C03646=1209.159,-22.656,-41.537,-179.909,5.502,148.937
C03647=1209.154,-22.387,-41.552,-179.907,5.502,148.936
C03648=1209.149,-22.137,-41.565,-179.904,5.503,148.936
C03649=1209.144,-21.888,-41.578,-179.901,5.503,148.935
C03650=1209.139,-21.638,-41.590,-179.899,5.503,148.934
C03651=1209.134,-21.388,-41.605,-179.897,5.503,148.934
C03652=1209.128,-21.139,-41.617,-179.894,5.504,148.933
C03653=1209.123,-20.889,-41.631,-179.891,5.504,148.932
C03654=1209.118,-20.640,-41.644,-179.889,5.504,148.932
C03655=1209.113,-20.390,-41.658,-179.887,5.505,148.931
C03656=1209.108,-20.140,-41.670,-179.884,5.505,148.930
C03657=1209.103,-19.890,-41.684,-179.882,5.506,148.930
C03658=1209.098,-19.641,-41.697,-179.880,5.505,148.929
C03659=1209.092,-19.392,-41.710,-179.877,5.506,148.928
C03660=1209.088,-19.142,-41.723,-179.874,5.506,148.928
C03661=1209.082,-18.893,-41.737,-179.872,5.507,148.927
C03662=1209.077,-18.643,-41.750,-179.870,5.507,148.926
C03663=1209.072,-18.393,-41.764,-179.867,5.507,148.926
C03664=1209.067,-18.144,-41.777,-179.864,5.508,148.925
C03665=1209.062,-17.894,-41.790,-179.862,5.508,148.924
C03666=1209.057,-17.644,-41.803,-179.860,5.508,148.924
C03667=1209.051,-17.395,-41.817,-179.857,5.509,148.923
C03668=1209.047,-17.145,-41.830,-179.855,5.509,148.922
C03669=1209.041,-16.896,-41.844,-179.852,5.510,148.922
C03670=1209.037,-16.646,-41.857,-179.850,5.509,148.921
C03671=1209.031,-16.396,-41.870,-179.847,5.510,148.920
C03672=1209.027,-16.147,-41.884,-179.845,5.510,148.920
C03673=1209.021,-15.897,-41.897,-179.842,5.511,148.919
C03674=1209.017,-15.648,-41.911,-179.840,5.510,148.918
C03675=1209.011,-15.398,-41.924,-179.838,5.511,148.918
C03676=1209.006,-15.149,-41.938,-179.835,5.512,148.917
C03677=1209.001,-14.899,-41.951,-179.832,5.512,148.916
C03678=1208.996,-14.650,-41.965,-179.830,5.512,148.916
C03679=1208.991,-14.400,-41.978,-179.828,5.512,148.915
C03680=1208.985,-14.150,-41.991,-179.825,5.513,148.914
C03681=1208.980,-13.900,-42.006,-179.822,5.513,148.914
C03682=1208.975,-13.651,-42.018,-179.820,5.514,148.913
C03683=1208.970,-13.401,-42.033,-179.818,5.514,148.912
C03684=1208.966,-13.153,-42.046,-179.815,5.514,148.911
C03685=1208.960,-12.902,-42.059,-179.813,5.515,148.911
C03686=1208.955,-12.653,-42.073,-179.810,5.515,148.910
C03687=1208.950,-12.403,-42.086,-179.808,5.515,148.910
C03688=1208.945,-12.153,-42.101,-179.805,5.516,148.909
C03689=1208.939,-11.904,-42.114,-179.803,5.516,148.908
C03690=1208.935,-11.654,-42.127,-179.800,5.517,148.908
C03691=1208.929,-11.405,-42.141,-179.798,5.517,148.907
C03692=1208.924,-11.155,-42.155,-179.795,5.517,148.906
C03693=1208.920,-10.906,-42.169,-179.793,5.517,148.905
C03694=1208.914,-10.656,-42.182,-179.791,5.518,148.905
C03695=1208.909,-10.406,-42.196,-179.788,5.519,148.904
C03696=1208.904,-10.157,-42.209,-179.785,5.519,148.904
C03697=1208.899,-9.907,-42.223,-179.783,5.519,148.903
C03698=1208.894,-9.658,-42.237,-179.781,5.519,148.902
C03699=1208.889,-9.408,-42.250,-179.778,5.520,148.902
C03700=1208.884,-9.159,-42.264,-179.775,5.520,148.901
C03701=1208.878,-8.909,-42.277,-179.773,5.520,148.900
C03702=1208.874,-8.660,-42.291,-179.771,5.520,148.899
C03703=1208.869,-8.410,-42.305,-179.768,5.521,148.899
C03704=1208.863,-8.160,-42.318,-179.766,5.522,148.898
C03705=1208.858,-7.911,-42.333,-179.763,5.522,148.898
C03706=1208.854,-7.661,-42.346,-179.761,5.522,148.897
C03707=1208.849,-7.412,-42.360,-179.758,5.522,148.896
C03708=1208.843,-7.162,-42.374,-179.756,5.523,148.896
C03709=1208.839,-6.912,-42.388,-179.753,5.523,148.895
C03710=1208.834,-6.663,-42.401,-179.750,5.524,148.894
C03711=1208.828,-6.413,-42.415,-179.748,5.524,148.893
C03712=1208.823,-6.163,-42.429,-179.746,5.524,148.893
C03713=1208.818,-5.914,-42.443,-179.743,5.525,148.892
C03714=1208.814,-5.665,-42.457,-179.741,5.525,148.892
C03715=1208.808,-5.415,-42.470,-179.738,5.526,148.891
C03716=1208.803,-5.166,-42.484,-179.736,5.526,148.890
C03717=1208.798,-4.916,-42.499,-179.733,5.526,148.890
C03718=1208.793,-4.666,-42.513,-179.731,5.527,148.889
C03719=1208.788,-4.417,-42.526,-179.728,5.527,148.888
C03720=1208.783,-4.167,-42.540,-179.725,5.528,148.887
C03721=1208.778,-3.917,-42.554,-179.723,5.529,148.887
C03722=1208.772,-3.668,-42.568,-179.721,5.528,148.886
C03723=1208.767,-3.419,-42.582,-179.719,5.529,148.886
C03724=1208.763,-3.169,-42.596,-179.716,5.529,148.885
C03725=1208.757,-2.920,-42.609,-179.713,5.530,148.884
C03726=1208.752,-2.670,-42.623,-179.711,5.530,148.884
C03727=1208.747,-2.420,-42.638,-179.709,5.530,148.883
C03728=1208.742,-2.171,-42.652,-179.706,5.530,148.882
C03729=1208.737,-1.922,-42.666,-179.703,5.531,148.882
C03730=1208.732,-1.672,-42.680,-179.701,5.532,148.881
C03731=1208.728,-1.422,-42.694,-179.698,5.532,148.880
C03732=1208.723,-1.173,-42.708,-179.696,5.533,148.880
C03733=1208.717,-0.923,-42.721,-179.694,5.532,148.879
C03734=1208.712,-0.673,-42.736,-179.691,5.533,148.878
C03735=1208.707,-0.424,-42.750,-179.688,5.533,148.878
C03736=1208.701,-0.175,-42.764,-179.686,5.534,148.877
C03737=1208.696,0.075,-42.778,-179.683,5.534,148.876
C03738=1208.691,0.325,-42.792,-179.681,5.535,148.876
C03739=1208.687,0.574,-42.807,-179.679,5.535,148.875
C03740=1208.682,0.824,-42.821,-179.676,5.536,148.874
C03741=1208.676,1.073,-42.835,-179.674,5.536,148.874
C03742=1208.672,1.323,-42.849,-179.671,5.537,148.873
C03743=1208.667,1.572,-42.863,-179.668,5.537,148.872
C03744=1208.662,1.822,-42.877,-179.666,5.538,148.872
C03745=1208.656,2.071,-42.891,-179.663,5.537,148.871
C03746=1208.651,2.321,-42.905,-179.661,5.538,148.870
C03747=1208.646,2.570,-42.920,-179.659,5.539,148.870
C03748=1208.641,2.840,-42.935,-179.656,5.539,148.869
C03749=1208.636,3.109,-42.950,-179.653,5.539,148.868
C03750=1208.629,3.378,-42.965,-179.650,5.540,148.868
C03751=1208.624,3.646,-42.981,-179.648,5.540,148.867
C03752=1208.619,3.896,-42.995,-179.645,5.541,148.866
C03753=1208.614,4.146,-43.010,-179.642,5.541,148.865
C03754=1208.609,4.396,-43.024,-179.640,5.542,148.865
C03755=1208.604,4.645,-43.038,-179.638,5.542,148.864
C03756=1208.599,4.894,-43.052,-179.635,5.542,148.864
C03757=1208.594,5.144,-43.066,-179.633,5.543,148.863
C03758=1208.589,5.394,-43.081,-179.630,5.543,148.862
C03759=1208.584,5.643,-43.095,-179.627,5.544,148.862
C03760=1208.579,5.893,-43.109,-179.625,5.544,148.861
C03761=1208.574,6.142,-43.124,-179.623,5.544,148.860
C03762=1208.569,6.391,-43.138,-179.621,5.545,148.860
C03763=1208.564,6.641,-43.152,-179.618,5.545,148.859
C03764=1208.559,6.891,-43.167,-179.615,5.546,148.858
C03765=1208.554,7.140,-43.181,-179.613,5.546,148.858
C03766=1208.549,7.390,-43.195,-179.610,5.547,148.857
C03767=1208.544,7.639,-43.210,-179.607,5.547,148.856
C03768=1208.539,7.889,-43.225,-179.605,5.548,148.856
C03769=1208.534,8.139,-43.239,-179.603,5.548,148.855
C03770=1208.529,8.388,-43.253,-179.600,5.549,148.854
C03771=1208.523,8.638,-43.268,-179.598,5.549,148.854
C03772=1208.518,8.887,-43.283,-179.595,5.550,148.853
C03773=1208.513,9.136,-43.297,-179.592,5.550,148.852
C03774=1208.508,9.386,-43.311,-179.590,5.551,148.852
C03775=1208.503,9.636,-43.325,-179.587,5.551,148.851
C03776=1208.498,9.886,-43.340,-179.585,5.551,148.850
C03777=1208.494,10.135,-43.355,-179.583,5.552,148.850
C03778=1208.489,10.384,-43.369,-179.580,5.552,148.849
C03779=1208.483,10.634,-43.384,-179.578,5.553,148.849
C03780=1208.478,10.883,-43.399,-179.575,5.553,148.848
C03781=1208.473,11.132,-43.413,-179.572,5.554,148.847
C03782=1208.468,11.382,-43.427,-179.570,5.554,148.846
C03783=1208.463,11.632,-43.441,-179.567,5.555,148.846
C03784=1208.458,11.881,-43.456,-179.565,5.555,148.845
C03785=1208.453,12.131,-43.471,-179.563,5.555,148.845
C03786=1208.448,12.381,-43.485,-179.560,5.556,148.844
C03787=1208.443,12.630,-43.500,-179.557,5.556,148.843
C03788=1208.438,12.880,-43.515,-179.555,5.557,148.843
C03789=1208.433,13.129,-43.529,-179.552,5.557,148.842
C03790=1208.428,13.379,-43.545,-179.550,5.558,148.841
C03791=1208.423,13.628,-43.559,-179.547,5.558,148.841
C03792=1208.418,13.878,-43.573,-179.545,5.559,148.840
C03793=1208.413,14.127,-43.588,-179.543,5.559,148.839
C03794=1208.408,14.377,-43.603,-179.540,5.560,148.839
C03795=1208.402,14.626,-43.618,-179.537,5.560,148.838
C03796=1208.397,14.875,-43.632,-179.535,5.561,148.837
C03797=1208.392,15.125,-43.646,-179.532,5.561,148.837
C03798=1208.387,15.374,-43.662,-179.529,5.562,148.836
C03799=1208.382,15.624,-43.676,-179.527,5.562,148.836
C03800=1208.377,15.873,-43.691,-179.525,5.563,148.835
C03801=1208.372,16.123,-43.705,-179.522,5.563,148.834
C03802=1208.367,16.372,-43.721,-179.519,5.564,148.833
C03803=1208.362,16.622,-43.735,-179.517,5.564,148.833
C03804=1208.357,16.871,-43.750,-179.515,5.564,148.832
C03805=1208.353,17.121,-43.764,-179.512,5.565,148.832
C03806=1208.347,17.370,-43.780,-179.510,5.566,148.831
C03807=1208.342,17.620,-43.794,-179.507,5.566,148.830
C03808=1208.338,17.869,-43.809,-179.504,5.567,148.830
C03809=1208.332,18.119,-43.824,-179.502,5.567,148.829
C03810=1208.327,18.368,-43.839,-179.499,5.568,148.828
C03811=1208.323,18.619,-43.854,-179.497,5.568,148.828
C03812=1208.317,18.868,-43.869,-179.494,5.569,148.827
C03813=1208.312,19.118,-43.884,-179.492,5.570,148.826
C03814=1208.308,19.367,-43.899,-179.490,5.569,148.826
C03815=1208.302,19.617,-43.914,-179.487,5.570,148.825
C03816=1208.297,19.866,-43.929,-179.484,5.570,148.824
C03817=1208.292,20.116,-43.943,-179.482,5.571,148.824
C03818=1208.287,20.365,-43.958,-179.480,5.572,148.823
C03819=1208.282,20.614,-43.973,-179.477,5.572,148.823
C03820=1208.277,20.864,-43.988,-179.474,5.573,148.822
C03821=1208.272,21.113,-44.003,-179.472,5.573,148.821
C03822=1208.267,21.363,-44.018,-179.469,5.574,148.821
C03823=1208.262,21.612,-44.033,-179.466,5.574,148.820
C03824=1208.257,21.861,-44.048,-179.464,5.575,148.819
C03825=1208.251,22.111,-44.063,-179.462,5.576,148.819
C03826=1208.247,22.361,-44.078,-179.459,5.576,148.818
C03827=1208.243,22.610,-44.093,-179.457,5.576,148.817
C03828=1208.237,22.860,-44.108,-179.454,5.577,148.817
C03829=1208.232,23.109,-44.123,-179.452,5.577,148.816
C03830=1208.227,23.359,-44.139,-179.449,5.578,148.815
C03831=1208.222,23.609,-44.153,-179.447,5.578,148.815
C03832=1208.217,23.858,-44.169,-179.444,5.579,148.814
C03833=1208.212,24.107,-44.184,-179.441,5.579,148.814
C03834=1208.207,24.356,-44.199,-179.439,5.580,148.813
C03835=1208.202,24.606,-44.214,-179.436,5.581,148.812
C03836=1208.197,24.856,-44.230,-179.433,5.581,148.811
C03837=1208.192,25.105,-44.245,-179.431,5.582,148.811
C03838=1208.187,25.355,-44.260,-179.429,5.582,148.810
C03839=1208.182,25.604,-44.274,-179.426,5.583,148.810
C03840=1208.177,25.854,-44.290,-179.423,5.584,148.809
C03841=1208.172,26.103,-44.305,-179.421,5.584,148.808
C03842=1208.167,26.352,-44.321,-179.418,5.585,148.808
C03843=1208.162,26.603,-44.335,-179.417,5.585,148.807
C03844=1208.157,26.852,-44.351,-179.414,5.585,148.806
C03845=1208.152,27.101,-44.366,-179.411,5.586,148.806
C03846=1208.147,27.351,-44.381,-179.409,5.586,148.805
C03847=1208.142,27.600,-44.396,-179.406,5.587,148.804
C03848=1208.136,27.850,-44.411,-179.403,5.587,148.804
C03849=1208.132,28.099,-44.426,-179.401,5.588,148.803
C03850=1208.127,28.349,-44.442,-179.398,5.589,148.803
C03851=1208.122,28.598,-44.457,-179.396,5.589,148.802
C03852=1208.117,28.867,-44.474,-179.393,5.590,148.801
C03853=1208.111,29.136,-44.490,-179.391,5.590,148.801
C03854=1208.106,29.404,-44.507,-179.388,5.591,148.800
C03855=1208.100,29.673,-44.523,-179.385,5.592,148.799
C03856=1208.095,29.922,-44.539,-179.382,5.593,148.799
C03857=1208.091,30.172,-44.554,-179.379,5.593,148.798
C03858=1208.085,30.421,-44.570,-179.377,5.593,148.797
C03859=1208.081,30.671,-44.585,-179.375,5.594,148.797
C03860=1208.075,30.920,-44.600,-179.373,5.594,148.796
C03861=1208.070,31.169,-44.616,-179.370,5.595,148.795
C03862=1208.066,31.419,-44.631,-179.367,5.595,148.795
C03863=1208.061,31.669,-44.647,-179.365,5.596,148.794
C03864=1208.055,31.918,-44.662,-179.362,5.596,148.793
C03865=1208.050,32.167,-44.677,-179.360,5.597,148.793
C03866=1208.046,32.417,-44.693,-179.357,5.598,148.792
C03867=1208.041,32.666,-44.708,-179.355,5.598,148.792
C03868=1208.036,32.916,-44.724,-179.352,5.599,148.791
C03869=1208.030,33.165,-44.740,-179.349,5.599,148.790
C03870=1208.026,33.415,-44.755,-179.347,5.600,148.790
C03871=1208.021,33.664,-44.770,-179.344,5.601,148.789
C03872=1208.015,33.914,-44.786,-179.342,5.601,148.788
C03873=1208.010,34.163,-44.802,-179.339,5.602,148.788
C03874=1208.006,34.413,-44.817,-179.337,5.602,148.787
C03875=1208.001,34.662,-44.833,-179.334,5.603,148.786
C03876=1207.995,34.912,-44.848,-179.332,5.604,148.786
C03877=1207.991,35.161,-44.863,-179.329,5.604,148.785
C03878=1207.986,35.411,-44.879,-179.326,5.605,148.785
C03879=1207.980,35.660,-44.895,-179.324,5.605,148.784
C03880=1207.975,35.910,-44.910,-179.321,5.606,148.783
C03881=1207.971,36.159,-44.926,-179.319,5.607,148.783
C03882=1207.966,36.408,-44.942,-179.316,5.607,148.782
C03883=1207.961,36.658,-44.958,-179.314,5.608,148.781
C03884=1207.956,36.908,-44.974,-179.311,5.608,148.781
C03885=1207.951,37.157,-44.989,-179.308,5.609,148.780
C03886=1207.946,37.406,-45.004,-179.306,5.610,148.780
C03887=1207.941,37.656,-45.020,-179.304,5.610,148.779
C03888=1207.936,37.906,-45.036,-179.301,5.611,148.778
C03889=1207.931,38.154,-45.051,-179.298,5.612,148.778
C03890=1207.926,38.404,-45.067,-179.296,5.612,148.777
C03891=1207.921,38.654,-45.083,-179.294,5.613,148.777
C03892=1207.916,38.903,-45.098,-179.291,5.613,148.776
C03893=1207.910,39.153,-45.114,-179.288,5.614,148.775
C03894=1207.906,39.402,-45.131,-179.286,5.615,148.775
C03895=1207.901,39.651,-45.146,-179.283,5.615,148.774
C03896=1207.896,39.901,-45.162,-179.281,5.616,148.773
C03897=1207.891,40.151,-45.177,-179.278,5.617,148.773
C03898=1207.886,40.399,-45.194,-179.276,5.617,148.772
C03899=1207.881,40.650,-45.210,-179.273,5.618,148.771
C03900=1207.876,40.899,-45.225,-179.270,5.618,148.771
C03901=1207.871,41.148,-45.240,-179.268,5.619,148.770
C03902=1207.867,41.397,-45.257,-179.265,5.620,148.770
C03903=1207.861,41.647,-45.272,-179.263,5.620,148.769
C03904=1207.856,41.897,-45.288,-179.260,5.621,148.768
C03905=1207.851,42.146,-45.305,-179.258,5.622,148.768
C03906=1207.846,42.395,-45.320,-179.255,5.622,148.767
C03907=1207.841,42.645,-45.336,-179.253,5.623,148.766
C03908=1207.836,42.894,-45.352,-179.250,5.623,148.766
C03909=1207.831,43.144,-45.368,-179.248,5.624,148.765
C03910=1207.827,43.393,-45.383,-179.245,5.625,148.765
C03911=1207.822,43.642,-45.400,-179.243,5.625,148.764
C03912=1207.817,43.892,-45.416,-179.240,5.626,148.763
C03913=1207.811,44.142,-45.431,-179.237,5.627,148.763
C03914=1207.807,44.391,-45.448,-179.234,5.628,148.762
C03915=1207.801,44.640,-45.464,-179.232,5.628,148.762
C03916=1207.796,44.889,-45.480,-179.229,5.629,148.761
C03917=1207.792,45.139,-45.496,-179.227,5.630,148.760
C03918=1207.786,45.389,-45.511,-179.224,5.630,148.760
C03919=1207.782,45.638,-45.528,-179.222,5.631,148.759
C03920=1207.776,45.888,-45.544,-179.219,5.632,148.758
C03921=1207.772,46.137,-45.560,-179.217,5.632,148.758
C03922=1207.767,46.386,-45.576,-179.214,5.633,148.757
C03923=1207.762,46.636,-45.593,-179.211,5.633,148.756
C03924=1207.757,46.885,-45.608,-179.209,5.634,148.756
C03925=1207.752,47.135,-45.625,-179.207,5.635,148.755
C03926=1207.747,47.384,-45.640,-179.204,5.635,148.755
C03927=1207.742,47.633,-45.657,-179.201,5.636,148.754
C03928=1207.737,47.883,-45.673,-179.199,5.637,148.753
C03929=1207.732,48.132,-45.689,-179.197,5.637,148.753
C03930=1207.727,48.382,-45.705,-179.194,5.638,148.752
C03931=1207.722,48.631,-45.721,-179.191,5.638,148.751
C03932=1207.717,48.881,-45.737,-179.189,5.639,148.751
C03933=1207.712,49.130,-45.753,-179.187,5.640,148.750
C03934=1207.707,49.380,-45.769,-179.183,5.641,148.750
C03935=1207.702,49.629,-45.786,-179.181,5.642,148.749
C03936=1207.698,49.878,-45.802,-179.179,5.642,148.749
C03937=1207.693,50.128,-45.818,-179.176,5.643,148.748
C03938=1207.688,50.377,-45.835,-179.173,5.644,148.747
C03939=1207.682,50.627,-45.851,-179.171,5.644,148.747
C03940=1207.677,50.876,-45.868,-179.168,5.645,148.746
C03941=1207.673,51.126,-45.884,-179.166,5.646,148.745
C03942=1207.667,51.375,-45.900,-179.163,5.646,148.745
C03943=1207.663,51.625,-45.916,-179.161,5.647,148.744
C03944=1207.658,51.873,-45.933,-179.158,5.647,148.743
C03945=1207.653,52.123,-45.949,-179.156,5.648,148.743
C03946=1207.648,52.372,-45.965,-179.153,5.649,148.742
C03947=1207.644,52.622,-45.982,-179.151,5.649,148.742
C03948=1207.637,52.871,-45.998,-179.147,5.651,148.741
C03949=1207.633,53.121,-46.015,-179.145,5.651,148.741
C03950=1207.628,53.370,-46.031,-179.143,5.652,148.740
C03951=1207.623,53.620,-46.047,-179.140,5.653,148.739
C03952=1207.619,53.869,-46.063,-179.137,5.653,148.739
C03953=1207.613,54.118,-46.080,-179.135,5.654,148.738
C03954=1207.608,54.368,-46.097,-179.132,5.655,148.737
C03955=1207.603,54.617,-46.113,-179.130,5.655,148.737
C03956=1207.598,54.886,-46.131,-179.127,5.656,148.736
C03957=1207.593,55.154,-46.148,-179.124,5.657,148.735
C03958=1207.588,55.423,-46.166,-179.121,5.658,148.735
C03959=1207.582,55.691,-46.184,-179.119,5.658,148.734
C03960=1207.577,55.941,-46.200,-179.117,5.659,148.734
C03961=1207.572,56.190,-46.216,-179.114,5.660,148.733
C03962=1207.568,56.439,-46.233,-179.111,5.660,148.732
C03963=1207.562,56.689,-46.250,-179.109,5.661,148.732
C03964=1207.557,56.938,-46.267,-179.106,5.662,148.731
C03965=1207.553,57.187,-46.283,-179.103,5.663,148.731
C03966=1207.548,57.437,-46.299,-179.101,5.663,148.730
C03967=1207.542,57.687,-46.316,-179.098,5.664,148.729
C03968=1207.538,57.936,-46.333,-179.096,5.665,148.729
C03969=1207.533,58.185,-46.349,-179.093,5.665,148.728
C03970=1207.528,58.434,-46.366,-179.091,5.666,148.728
C03971=1207.523,58.684,-46.383,-179.088,5.667,148.727
C03972=1207.518,58.933,-46.399,-179.086,5.667,148.726
C03973=1207.513,59.182,-46.416,-179.083,5.669,148.726
C03974=1207.508,59.433,-46.433,-179.080,5.669,148.725
C03975=1207.503,59.682,-46.449,-179.078,5.670,148.725
C03976=1207.498,59.931,-46.466,-179.075,5.671,148.724
C03977=1207.493,60.181,-46.483,-179.073,5.671,148.723
C03978=1207.488,60.430,-46.499,-179.070,5.672,148.723
C03979=1207.484,60.679,-46.516,-179.068,5.673,148.722
C03980=1207.478,60.929,-46.533,-179.065,5.673,148.722
C03981=1207.473,61.178,-46.549,-179.063,5.674,148.721
C03982=1207.469,61.427,-46.566,-179.060,5.676,148.720
C03983=1207.464,61.677,-46.583,-179.057,5.676,148.720
C03984=1207.459,61.926,-46.600,-179.055,5.677,148.719
C03985=1207.454,62.175,-46.616,-179.052,5.677,148.718
C03986=1207.449,62.425,-46.634,-179.050,5.678,148.718
C03987=1207.444,62.675,-46.650,-179.047,5.679,148.717
C03988=1207.439,62.924,-46.667,-179.045,5.679,148.717
C03989=1207.434,63.173,-46.684,-179.042,5.681,148.716
C03990=1207.430,63.423,-46.700,-179.039,5.682,148.716
C03991=1207.424,63.672,-46.717,-179.037,5.682,148.715
C03992=1207.419,63.921,-46.734,-179.034,5.683,148.714
C03993=1207.414,64.171,-46.751,-179.032,5.684,148.714
C03994=1207.410,64.420,-46.769,-179.029,5.684,148.713
C03995=1207.405,64.669,-46.785,-179.027,5.685,148.713
C03996=1207.400,64.918,-46.802,-179.024,5.686,148.712
C03997=1207.395,65.168,-46.819,-179.021,5.687,148.711
C03998=1207.390,65.418,-46.836,-179.019,5.688,148.711
C03999=1207.385,65.667,-46.852,-179.016,5.688,148.710
C04000=1207.380,65.916,-46.870,-179.014,5.689,148.710
C04001=1207.375,66.166,-46.886,-179.011,5.690,148.709
C04002=1207.370,66.415,-46.904,-179.008,5.690,148.708
C04003=1207.366,66.664,-46.921,-179.006,5.692,148.708
C04004=1207.361,66.913,-46.937,-179.003,5.693,148.707
C04005=1207.355,67.163,-46.955,-179.001,5.693,148.707
C04006=1207.351,67.413,-46.971,-178.998,5.694,148.706
C04007=1207.346,67.662,-46.989,-178.996,5.695,148.706
C04008=1207.342,67.911,-47.006,-178.993,5.695,148.705
C04009=1207.336,68.160,-47.023,-178.990,5.696,148.704
C04010=1207.331,68.410,-47.039,-178.988,5.697,148.704
C04011=1207.326,68.660,-47.057,-178.985,5.698,148.703
C04012=1207.321,68.909,-47.075,-178.982,5.699,148.702
C04013=1207.317,69.158,-47.091,-178.980,5.699,148.702
C04014=1207.311,69.407,-47.108,-178.978,5.700,148.701
C04015=1207.306,69.657,-47.125,-178.975,5.701,148.701
C04016=1207.301,69.906,-47.143,-178.972,5.702,148.700
C04017=1207.297,70.155,-47.160,-178.970,5.703,148.700
C04018=1207.292,70.405,-47.177,-178.967,5.703,148.699
C04019=1207.288,70.654,-47.194,-178.965,5.704,148.698
C04020=1207.282,70.903,-47.211,-178.962,5.705,148.698
C04021=1207.277,71.153,-47.228,-178.960,5.705,148.697
C04022=1207.272,71.402,-47.246,-178.957,5.707,148.697
C04023=1207.267,71.652,-47.263,-178.954,5.708,148.696
C04024=1207.263,71.901,-47.280,-178.952,5.708,148.695
C04025=1207.258,72.150,-47.298,-178.949,5.709,148.695
C04026=1207.253,72.400,-47.315,-178.947,5.710,148.694
C04027=1207.248,72.650,-47.332,-178.944,5.711,148.694
C04028=1207.243,72.898,-47.349,-178.941,5.712,148.693
C04029=1207.237,73.148,-47.367,-178.939,5.713,148.693
C04030=1207.233,73.397,-47.384,-178.936,5.713,148.692
C04031=1207.228,73.647,-47.401,-178.934,5.714,148.691
C04032=1207.223,73.896,-47.418,-178.931,5.716,148.691
C04033=1207.219,74.145,-47.436,-178.928,5.716,148.690
C04034=1207.213,74.395,-47.453,-178.926,5.717,148.690
C04035=1207.208,74.644,-47.471,-178.924,5.718,148.689
C04036=1207.204,74.894,-47.488,-178.921,5.718,148.688
C04037=1207.198,75.142,-47.505,-178.918,5.719,148.688
C04038=1207.193,75.392,-47.523,-178.916,5.720,148.687
C04039=1207.189,75.641,-47.540,-178.913,5.721,148.687
C04040=1207.184,75.891,-47.557,-178.910,5.722,148.686
C04041=1207.179,76.140,-47.575,-178.908,5.723,148.686
C04042=1207.174,76.389,-47.592,-178.906,5.723,148.685
C04043=1207.169,76.638,-47.610,-178.902,5.724,148.684
C04044=1207.164,76.888,-47.627,-178.900,5.725,148.684
C04045=1207.159,77.137,-47.645,-178.898,5.726,148.683
C04046=1207.155,77.387,-47.662,-178.895,5.727,148.683
C04047=1207.150,77.636,-47.680,-178.892,5.728,148.682
C04048=1207.145,77.885,-47.698,-178.890,5.729,148.681
C04049=1207.140,78.135,-47.715,-178.887,5.729,148.681
C04050=1207.136,78.384,-47.732,-178.885,5.730,148.680
C04051=1207.130,78.634,-47.750,-178.882,5.731,148.680
C04052=1207.126,78.883,-47.768,-178.879,5.732,148.679
C04053=1207.121,79.132,-47.786,-178.877,5.733,148.679
C04054=1207.115,79.382,-47.803,-178.874,5.734,148.678
C04055=1207.111,79.631,-47.820,-178.872,5.735,148.678
C04056=1207.106,79.881,-47.838,-178.869,5.736,148.677
C04057=1207.101,80.130,-47.856,-178.866,5.737,148.676
C04058=1207.096,80.379,-47.874,-178.864,5.738,148.676
C04059=1207.091,80.629,-47.891,-178.862,5.738,148.675
C04060=1207.085,80.896,-47.910,-178.858,5.740,148.675
C04061=1207.080,81.164,-47.929,-178.856,5.740,148.674
C04062=1207.076,81.433,-47.947,-178.853,5.741,148.673
C04063=1207.070,81.701,-47.967,-178.850,5.742,148.673
C04064=1207.065,81.951,-47.984,-178.848,5.743,148.672
C04065=1207.060,82.200,-48.002,-178.845,5.744,148.672
C04066=1207.055,82.449,-48.020,-178.843,5.745,148.671
C04067=1207.051,82.699,-48.038,-178.840,5.746,148.670
C04068=1207.045,82.948,-48.055,-178.837,5.746,148.670
C04069=1207.040,83.198,-48.073,-178.835,5.747,148.669
C04070=1207.035,83.447,-48.091,-178.833,5.748,148.669
C04071=1207.031,83.696,-48.109,-178.829,5.749,148.668
C04072=1207.026,83.945,-48.127,-178.827,5.750,148.668
C04073=1207.021,84.195,-48.144,-178.825,5.751,148.667
C04074=1207.017,84.444,-48.162,-178.822,5.752,148.667
C04075=1207.012,84.694,-48.180,-178.819,5.753,148.666
C04076=1207.007,84.943,-48.198,-178.817,5.754,148.665
C04077=1207.002,85.192,-48.216,-178.814,5.755,148.665
C04078=1206.997,85.442,-48.233,-178.812,5.755,148.664
C04079=1206.992,85.691,-48.251,-178.809,5.757,148.664
C04080=1206.987,85.940,-48.269,-178.807,5.758,148.663
C04081=1206.982,86.189,-48.287,-178.804,5.758,148.662
C04082=1206.977,86.438,-48.305,-178.801,5.760,148.662
C04083=1206.972,86.688,-48.323,-178.799,5.760,148.661
C04084=1206.967,86.937,-48.341,-178.796,5.761,148.661
C04085=1206.963,87.187,-48.360,-178.794,5.762,148.660
C04086=1206.958,87.436,-48.378,-178.791,5.763,148.660
C04087=1206.953,87.685,-48.396,-178.788,5.764,148.659
C04088=1206.948,87.935,-48.413,-178.786,5.765,148.659
C04089=1206.943,88.184,-48.431,-178.783,5.765,148.658
C04090=1206.938,88.433,-48.449,-178.781,5.767,148.658
C04091=1206.933,88.682,-48.467,-178.778,5.768,148.657
C04092=1206.928,88.932,-48.485,-178.776,5.769,148.656
C04093=1206.924,89.181,-48.503,-178.773,5.769,148.656
C04094=1206.919,89.431,-48.521,-178.770,5.771,148.655
C04095=1206.914,89.680,-48.539,-178.768,5.772,148.655
C04096=1206.909,89.929,-48.557,-178.765,5.772,148.654
C04097=1206.904,90.178,-48.575,-178.763,5.774,148.654
C04098=1206.900,90.427,-48.593,-178.760,5.774,148.653
C04099=1206.895,90.676,-48.611,-178.757,5.775,148.652
C04100=1206.890,90.926,-48.629,-178.755,5.776,148.652
C04101=1206.885,91.176,-48.648,-178.752,5.777,148.651
C04102=1206.880,91.424,-48.667,-178.750,5.778,148.651
C04103=1206.875,91.674,-48.685,-178.747,5.779,148.650
C04104=1206.870,91.923,-48.703,-178.744,5.780,148.650
C04105=1206.866,92.173,-48.721,-178.742,5.781,148.649
C04106=1206.861,92.422,-48.739,-178.739,5.782,148.649
C04107=1206.856,92.671,-48.757,-178.737,5.784,148.648
C04108=1206.851,92.920,-48.775,-178.734,5.784,148.647
C04109=1206.846,93.170,-48.793,-178.731,5.785,148.647
C04110=1206.841,93.420,-48.812,-178.729,5.786,148.646
C04111=1206.837,93.668,-48.830,-178.726,5.787,148.646
C04112=1206.832,93.917,-48.848,-178.724,5.788,148.645
C04113=1206.827,94.166,-48.866,-178.721,5.789,148.645
C04114=1206.822,94.416,-48.885,-178.718,5.790,148.644
C04115=1206.817,94.666,-48.903,-178.716,5.791,148.644
C04116=1206.812,94.915,-48.921,-178.713,5.791,148.643
C04117=1206.807,95.164,-48.940,-178.711,5.793,148.643
C04118=1206.802,95.413,-48.958,-178.708,5.794,148.642
C04119=1206.798,95.663,-48.976,-178.706,5.795,148.641
C04120=1206.792,95.912,-48.995,-178.703,5.796,148.641
C04121=1206.788,96.161,-49.014,-178.700,5.797,148.640
C04122=1206.783,96.410,-49.032,-178.698,5.798,148.640
C04123=1206.779,96.660,-49.050,-178.695,5.798,148.639
C04124=1206.774,96.909,-49.068,-178.693,5.800,148.639
C04125=1206.768,97.158,-49.087,-178.690,5.801,148.638
C04126=1206.764,97.408,-49.106,-178.688,5.801,148.638
C04127=1206.759,97.657,-49.124,-178.685,5.803,148.637
C04128=1206.754,97.906,-49.143,-178.682,5.804,148.637
C04129=1206.749,98.155,-49.161,-178.680,5.804,148.636
C04130=1206.745,98.405,-49.179,-178.677,5.806,148.635
C04131=1206.740,98.654,-49.197,-178.675,5.807,148.635
C04132=1206.734,98.903,-49.216,-178.672,5.807,148.634
C04133=1206.730,99.153,-49.235,-178.669,5.809,148.634
C04134=1206.725,99.401,-49.253,-178.667,5.810,148.633
C04135=1206.720,99.651,-49.272,-178.664,5.811,148.633
C04136=1206.715,99.901,-49.290,-178.661,5.812,148.632
C04137=1206.711,100.149,-49.309,-178.659,5.813,148.632
C04138=1206.705,100.399,-49.328,-178.657,5.814,148.631
C04139=1206.701,100.648,-49.347,-178.653,5.815,148.630
C04140=1206.696,100.897,-49.365,-178.651,5.816,148.630
C04141=1206.691,101.146,-49.383,-178.649,5.816,148.629
C04142=1206.687,101.396,-49.402,-178.646,5.818,148.629
C04143=1206.682,101.645,-49.420,-178.643,5.819,148.628
C04144=1206.676,101.894,-49.440,-178.641,5.821,148.628
C04145=1206.672,102.144,-49.458,-178.638,5.821,148.627
C04146=1206.667,102.392,-49.477,-178.636,5.822,148.627
C04147=1206.662,102.642,-49.495,-178.633,5.823,148.626
C04148=1206.658,102.891,-49.514,-178.631,5.824,148.626
C04149=1206.652,103.140,-49.533,-178.628,5.825,148.625
C04150=1206.648,103.390,-49.552,-178.625,5.826,148.625
C04151=1206.643,103.639,-49.570,-178.623,5.827,148.624
C04152=1206.638,103.888,-49.589,-178.620,5.828,148.623
C04153=1206.634,104.138,-49.608,-178.617,5.830,148.623
C04154=1206.628,104.386,-49.627,-178.615,5.830,148.622
C04155=1206.623,104.636,-49.645,-178.613,5.831,148.622
C04156=1206.619,104.885,-49.664,-178.609,5.833,148.621
C04157=1206.614,105.134,-49.682,-178.607,5.834,148.621
C04158=1206.609,105.384,-49.702,-178.604,5.835,148.620
C04159=1206.604,105.633,-49.721,-178.602,5.836,148.620
C04160=1206.600,105.882,-49.739,-178.599,5.837,148.619
C04161=1206.595,106.131,-49.758,-178.597,5.838,148.619
C04162=1206.590,106.380,-49.777,-178.594,5.839,148.618
C04163=1206.585,106.630,-49.796,-178.592,5.840,148.618
C04164=1206.579,106.898,-49.817,-178.589,5.841,148.617
C04165=1206.575,107.167,-49.837,-178.585,5.843,148.617
C04166=1206.569,107.435,-49.857,-178.583,5.843,148.616
C04167=1206.564,107.703,-49.877,-178.580,5.845,148.615
C04168=1206.560,107.953,-49.896,-178.578,5.846,148.615
C04169=1206.554,108.202,-49.916,-178.575,5.847,148.614
C04170=1206.550,108.451,-49.934,-178.572,5.848,148.614
C04171=1206.545,108.700,-49.953,-178.570,5.849,148.613
C04172=1206.540,108.950,-49.973,-178.567,5.850,148.613
C04173=1206.535,109.198,-49.992,-178.565,5.851,148.612
C04174=1206.530,109.449,-50.011,-178.562,5.852,148.612
C04175=1206.526,109.697,-50.029,-178.560,5.854,148.611
C04176=1206.521,109.947,-50.049,-178.557,5.854,148.611
C04177=1206.516,110.195,-50.068,-178.554,5.856,148.610
C04178=1206.511,110.445,-50.087,-178.552,5.857,148.610
C04179=1206.506,110.694,-50.106,-178.549,5.857,148.609
C04180=1206.502,110.944,-50.125,-178.546,5.859,148.609
C04181=1206.497,111.192,-50.144,-178.544,5.860,148.608
C04182=1206.493,111.442,-50.163,-178.541,5.861,148.608
C04183=1206.487,111.691,-50.182,-178.539,5.862,148.607
C04184=1206.482,111.941,-50.201,-178.536,5.864,148.606
C04185=1206.478,112.189,-50.220,-178.534,5.865,148.606
C04186=1206.473,112.439,-50.240,-178.531,5.865,148.605
C04187=1206.467,112.688,-50.259,-178.528,5.867,148.605
C04188=1206.463,112.937,-50.278,-178.526,5.868,148.604
C04189=1206.458,113.186,-50.297,-178.523,5.869,148.604
C04190=1206.453,113.435,-50.317,-178.520,5.870,148.603
C04191=1206.449,113.685,-50.335,-178.518,5.871,148.603
C04192=1206.444,113.934,-50.355,-178.515,5.872,148.602
C04193=1206.439,114.184,-50.374,-178.513,5.873,148.602
C04194=1206.434,114.432,-50.393,-178.510,5.875,148.601
C04195=1206.430,114.682,-50.413,-178.508,5.876,148.601
C04196=1206.424,114.931,-50.432,-178.504,5.877,148.600
C04197=1206.420,115.180,-50.452,-178.502,5.878,148.600
C04198=1206.416,115.430,-50.471,-178.500,5.879,148.599
C04199=1206.410,115.678,-50.490,-178.497,5.880,148.599
C04200=1206.405,115.928,-50.510,-178.495,5.881,148.598
C04201=1206.400,116.177,-50.529,-178.492,5.883,148.598
C04202=1206.396,116.426,-50.548,-178.490,5.884,148.597
C04203=1206.391,116.675,-50.567,-178.486,5.885,148.597
C04204=1206.386,116.925,-50.587,-178.484,5.886,148.596
C04205=1206.381,117.174,-50.607,-178.482,5.887,148.596
C04206=1206.377,117.423,-50.625,-178.479,5.888,148.595
C04207=1206.372,117.672,-50.645,-178.476,5.889,148.595
C04208=1206.367,117.922,-50.665,-178.474,5.891,148.594
C04209=1206.362,118.171,-50.684,-178.471,5.891,148.594
C04210=1206.357,118.420,-50.704,-178.468,5.893,148.593
C04211=1206.353,118.668,-50.723,-178.466,5.894,148.593
C04212=1206.348,118.918,-50.743,-178.463,5.895,148.592
C04213=1206.343,119.167,-50.762,-178.461,5.896,148.592
C04214=1206.338,119.416,-50.782,-178.458,5.898,148.591
C04215=1206.333,119.666,-50.801,-178.456,5.899,148.591
C04216=1206.328,119.915,-50.821,-178.453,5.899,148.590
C04217=1206.324,120.164,-50.840,-178.450,5.901,148.590
C04218=1206.319,120.413,-50.860,-178.448,5.902,148.589
C04219=1206.315,120.662,-50.880,-178.445,5.904,148.589
C04220=1206.309,120.911,-50.899,-178.442,5.904,148.588
C04221=1206.305,121.161,-50.919,-178.440,5.906,148.588
C04222=1206.300,121.410,-50.938,-178.438,5.907,148.587
C04223=1206.295,121.659,-50.958,-178.434,5.908,148.587
C04224=1206.290,121.908,-50.978,-178.432,5.909,148.586
C04225=1206.286,122.158,-50.997,-178.429,5.911,148.586
C04226=1206.281,122.406,-51.016,-178.427,5.912,148.585
C04227=1206.276,122.656,-51.036,-178.424,5.913,148.585
C04228=1206.272,122.905,-51.056,-178.422,5.914,148.584
C04229=1206.267,123.154,-51.076,-178.419,5.916,148.584
C04230=1206.261,123.403,-51.095,-178.416,5.916,148.583
C04231=1206.257,123.652,-51.116,-178.414,5.918,148.583
C04232=1206.252,123.902,-51.135,-178.411,5.919,148.582
C04233=1206.248,124.151,-51.155,-178.408,5.920,148.582
C04234=1206.242,124.400,-51.174,-178.406,5.921,148.581
C04235=1206.238,124.649,-51.195,-178.404,5.922,148.581
C04236=1206.233,124.899,-51.214,-178.401,5.924,148.580
C04237=1206.228,125.147,-51.234,-178.398,5.924,148.580
C04238=1206.223,125.397,-51.254,-178.396,5.926,148.579
C04239=1206.218,125.646,-51.274,-178.393,5.927,148.579
C04240=1206.214,125.895,-51.294,-178.390,5.929,148.578
C04241=1206.209,126.145,-51.314,-178.388,5.929,148.578
C04242=1206.204,126.394,-51.333,-178.385,5.931,148.577
C04243=1206.200,126.643,-51.353,-178.383,5.932,148.577
C04244=1206.195,126.892,-51.373,-178.380,5.933,148.576
C04245=1206.190,127.141,-51.393,-178.378,5.934,148.576
C04246=1206.185,127.390,-51.413,-178.375,5.936,148.575
C04247=1206.181,127.639,-51.433,-178.372,5.937,148.575
C04248=1206.176,127.888,-51.453,-178.370,5.938,148.574
C04249=1206.171,128.138,-51.472,-178.367,5.939,148.574
C04250=1206.167,128.387,-51.493,-178.364,5.941,148.573
C04251=1206.161,128.636,-51.512,-178.361,5.942,148.573
C04252=1206.157,128.885,-51.532,-178.359,5.943,148.572
C04253=1206.152,129.134,-51.552,-178.356,5.945,148.572
C04254=1206.148,129.383,-51.572,-178.354,5.946,148.571
C04255=1206.143,129.633,-51.593,-178.351,5.947,148.571
C04256=1206.138,129.882,-51.613,-178.349,5.948,148.570
C04257=1206.133,130.130,-51.633,-178.346,5.950,148.570
C04258=1206.128,130.380,-51.653,-178.344,5.951,148.569
C04259=1206.124,130.629,-51.673,-178.341,5.952,148.569
C04260=1206.119,130.878,-51.693,-178.338,5.953,148.568
C04261=1206.114,131.127,-51.713,-178.336,5.955,148.568
C04262=1206.109,131.377,-51.733,-178.333,5.955,148.567
C04263=1206.104,131.626,-51.753,-178.331,5.957,148.567
C04264=1206.099,131.874,-51.774,-178.328,5.958,148.566
C04265=1206.095,132.124,-51.793,-178.325,5.960,148.566
C04266=1206.090,132.373,-51.814,-178.323,5.961,148.566
C04267=1206.086,132.622,-51.834,-178.320,5.962,148.565
C04268=1206.080,132.891,-51.856,-178.317,5.964,148.565
C04269=1206.074,133.160,-51.877,-178.315,5.964,148.564
C04270=1206.070,133.428,-51.899,-178.312,5.966,148.564
C04271=1206.064,133.697,-51.921,-178.309,5.968,148.563
C04272=1206.060,133.946,-51.941,-178.307,5.969,148.563
C04273=1206.055,134.195,-51.962,-178.304,5.970,148.562
C04274=1206.051,134.444,-51.982,-178.301,5.972,148.562
C04275=1206.045,134.694,-52.002,-178.299,5.973,148.561
C04276=1206.041,134.943,-52.023,-178.296,5.974,148.561
C04277=1206.037,135.191,-52.043,-178.293,5.975,148.560
C04278=1206.032,135.441,-52.063,-178.290,5.977,148.559
C04279=1206.027,135.690,-52.084,-178.288,5.978,148.559
C04280=1206.022,135.939,-52.104,-178.285,5.979,148.559
C04281=1206.017,136.187,-52.124,-178.283,5.980,148.558
C04282=1206.012,136.437,-52.145,-178.280,5.982,148.558
C04283=1206.007,136.686,-52.165,-178.277,5.984,148.557
C04284=1206.003,136.935,-52.185,-178.275,5.984,148.557
C04285=1205.998,137.184,-52.205,-178.272,5.986,148.556
C04286=1205.993,137.433,-52.226,-178.270,5.987,148.556
C04287=1205.989,137.682,-52.247,-178.267,5.988,148.555
C04288=1205.984,137.931,-52.267,-178.265,5.989,148.555
C04289=1205.979,138.181,-52.287,-178.262,5.991,148.554
C04290=1205.974,138.430,-52.308,-178.259,5.993,148.554
C04291=1205.970,138.679,-52.328,-178.257,5.993,148.553
C04292=1205.965,138.928,-52.349,-178.254,5.995,148.553
C04293=1205.960,139.177,-52.369,-178.252,5.996,148.552
C04294=1205.955,139.427,-52.390,-178.249,5.998,148.552
C04295=1205.951,139.676,-52.411,-178.247,5.999,148.552
C04296=1205.946,139.925,-52.431,-178.244,6.000,148.551
C04297=1205.941,140.174,-52.452,-178.241,6.002,148.551
C04298=1205.937,140.423,-52.472,-178.239,6.003,148.550
C04299=1205.932,140.672,-52.493,-178.236,6.004,148.550
C04300=1205.927,140.921,-52.514,-178.234,6.005,148.549
C04301=1205.923,141.170,-52.534,-178.231,6.007,148.549
C04302=1205.917,141.419,-52.555,-178.228,6.008,148.548
C04303=1205.913,141.668,-52.576,-178.226,6.009,148.548
C04304=1205.908,141.917,-52.596,-178.223,6.011,148.548
C04305=1205.903,142.166,-52.617,-178.220,6.012,148.547
C04306=1205.898,142.416,-52.638,-178.218,6.014,148.547
C04307=1205.894,142.665,-52.658,-178.215,6.015,148.546
C04308=1205.889,142.913,-52.679,-178.212,6.016,148.545
C04309=1205.884,143.163,-52.700,-178.210,6.018,148.545
C04310=1205.880,143.412,-52.720,-178.208,6.019,148.545
C04311=1205.875,143.662,-52.741,-178.204,6.020,148.544
C04312=1205.871,143.911,-52.762,-178.202,6.022,148.544
C04313=1205.866,144.160,-52.783,-178.200,6.023,148.543
C04314=1205.861,144.409,-52.803,-178.197,6.025,148.543
C04315=1205.856,144.658,-52.824,-178.194,6.025,148.542
C04316=1205.852,144.906,-52.845,-178.192,6.027,148.542
C04317=1205.847,145.156,-52.866,-178.189,6.029,148.542
C04318=1205.842,145.405,-52.886,-178.186,6.030,148.541
C04319=1205.837,145.654,-52.907,-178.184,6.031,148.541
C04320=1205.832,145.903,-52.928,-178.181,6.033,148.540
C04321=1205.828,146.153,-52.949,-178.178,6.034,148.540
C04322=1205.823,146.401,-52.971,-178.176,6.036,148.539
C04323=1205.819,146.650,-52.991,-178.174,6.036,148.539
C04324=1205.814,146.900,-53.012,-178.171,6.038,148.538
C04325=1205.809,147.149,-53.032,-178.168,6.040,148.538
C04326=1205.804,147.397,-53.054,-178.166,6.041,148.537
C04327=1205.799,147.646,-53.075,-178.163,6.042,148.537
C04328=1205.795,147.895,-53.095,-178.160,6.044,148.536
C04329=1205.790,148.145,-53.117,-178.158,6.045,148.536
C04330=1205.786,148.394,-53.138,-178.155,6.047,148.536
C04331=1205.781,148.643,-53.159,-178.153,6.048,148.535
C04332=1205.776,148.892,-53.180,-178.150,6.049,148.535
C04333=1205.771,149.141,-53.200,-178.147,6.051,148.534
C04334=1205.766,149.390,-53.222,-178.145,6.052,148.534
C04335=1205.762,149.640,-53.243,-178.142,6.053,148.533
C04336=1205.757,149.889,-53.264,-178.139,6.055,148.533
C04337=1205.752,150.137,-53.285,-178.137,6.056,148.532
C04338=1205.747,150.387,-53.306,-178.134,6.058,148.532
C04339=1205.743,150.635,-53.327,-178.131,6.059,148.532
C04340=1205.738,150.884,-53.348,-178.129,6.060,148.531
C04341=1205.733,151.134,-53.370,-178.126,6.062,148.531
C04342=1205.729,151.382,-53.391,-178.124,6.064,148.530
C04343=1205.724,151.632,-53.412,-178.121,6.064,148.530
C04344=1205.719,151.880,-53.433,-178.118,6.066,148.529
C04345=1205.714,152.130,-53.454,-178.116,6.068,148.529
C04346=1205.710,152.379,-53.475,-178.114,6.069,148.529
C04347=1205.705,152.628,-53.497,-178.111,6.070,148.528
C04348=1205.700,152.877,-53.518,-178.108,6.072,148.528
C04349=1205.695,153.126,-53.539,-178.106,6.073,148.527
C04350=1205.691,153.375,-53.560,-178.103,6.075,148.527
C04351=1205.687,153.624,-53.582,-178.100,6.076,148.526
C04352=1205.681,153.873,-53.603,-178.098,6.077,148.526
C04353=1205.677,154.122,-53.624,-178.095,6.079,148.525
C04354=1205.673,154.372,-53.645,-178.092,6.081,148.525
C04355=1205.668,154.620,-53.667,-178.090,6.082,148.525
C04356=1205.663,154.870,-53.688,-178.087,6.083,148.524
C04357=1205.658,155.118,-53.709,-178.085,6.085,148.524
C04358=1205.653,155.368,-53.731,-178.082,6.086,148.523
C04359=1205.649,155.617,-53.752,-178.079,6.088,148.523
C04360=1205.644,155.865,-53.774,-178.077,6.089,148.522
C04361=1205.639,156.114,-53.795,-178.074,6.090,148.522
C04362=1205.635,156.364,-53.817,-178.072,6.092,148.522
C04363=1205.630,156.613,-53.838,-178.069,6.094,148.521
C04364=1205.625,156.862,-53.859,-178.067,6.095,148.521
C04365=1205.621,157.111,-53.881,-178.064,6.096,148.520
C04366=1205.616,157.360,-53.902,-178.061,6.098,148.520
C04367=1205.611,157.609,-53.923,-178.059,6.100,148.520
C04368=1205.607,157.858,-53.945,-178.056,6.101,148.519
C04369=1205.602,158.107,-53.966,-178.053,6.102,148.519
C04370=1205.597,158.356,-53.988,-178.051,6.104,148.518
C04371=1205.592,158.604,-54.010,-178.048,6.105,148.518
C04372=1205.587,158.873,-54.033,-178.045,6.107,148.517
C04373=1205.582,159.143,-54.056,-178.043,6.109,148.517
C04374=1205.577,159.411,-54.079,-178.040,6.110,148.516
C04375=1205.572,159.681,-54.103,-178.037,6.112,148.516
C04376=1205.568,159.930,-54.125,-178.034,6.114,148.515
C04377=1205.562,160.179,-54.146,-178.032,6.115,148.515
C04378=1205.557,160.428,-54.167,-178.029,6.116,148.514
C04379=1205.553,160.677,-54.189,-178.026,6.118,148.514
C04380=1205.548,160.926,-54.211,-178.024,6.120,148.514
C04381=1205.544,161.175,-54.233,-178.021,6.121,148.513
C04382=1205.539,161.424,-54.254,-178.019,6.122,148.513
C04383=1205.534,161.673,-54.276,-178.016,6.124,148.512
C04384=1205.530,161.922,-54.298,-178.013,6.126,148.512
C04385=1205.525,162.171,-54.320,-178.011,6.127,148.512
C04386=1205.521,162.420,-54.342,-178.008,6.128,148.511
C04387=1205.516,162.669,-54.363,-178.006,6.130,148.511
C04388=1205.511,162.918,-54.385,-178.003,6.131,148.510
C04389=1205.506,163.168,-54.406,-178.000,6.133,148.510
C04390=1205.501,163.416,-54.428,-177.998,6.134,148.510
C04391=1205.497,163.666,-54.450,-177.995,6.136,148.509
C04392=1205.492,163.914,-54.472,-177.993,6.137,148.509
C04393=1205.487,164.163,-54.493,-177.990,6.139,148.508
C04394=1205.483,164.412,-54.515,-177.987,6.140,148.508
C04395=1205.478,164.661,-54.537,-177.984,6.142,148.507
C04396=1205.474,164.910,-54.559,-177.982,6.143,148.507
C04397=1205.469,165.159,-54.581,-177.980,6.145,148.507
C04398=1205.465,165.408,-54.603,-177.977,6.147,148.506
C04399=1205.460,165.657,-54.625,-177.974,6.148,148.506
C04400=1205.455,165.907,-54.647,-177.972,6.149,148.505
C04401=1205.450,166.155,-54.669,-177.969,6.151,148.505
C04402=1205.446,166.405,-54.691,-177.966,6.153,148.505
C04403=1205.441,166.653,-54.713,-177.964,6.155,148.504
C04404=1205.436,166.902,-54.734,-177.962,6.156,148.504
C04405=1205.432,167.151,-54.756,-177.958,6.157,148.503
C04406=1205.427,167.400,-54.778,-177.956,6.159,148.503
C04407=1205.423,167.649,-54.800,-177.953,6.161,148.503
C04408=1205.417,167.898,-54.822,-177.951,6.162,148.502
C04409=1205.413,168.147,-54.844,-177.948,6.164,148.502
C04410=1205.408,168.396,-54.866,-177.946,6.165,148.501
C04411=1205.404,168.645,-54.889,-177.942,6.167,148.501
C04412=1205.399,168.893,-54.911,-177.940,6.169,148.500
C04413=1205.394,169.143,-54.933,-177.938,6.170,148.500
C04414=1205.389,169.392,-54.955,-177.935,6.171,148.500
C04415=1205.385,169.641,-54.977,-177.932,6.173,148.499
C04416=1205.380,169.890,-54.999,-177.930,6.175,148.499
C04417=1205.376,170.139,-55.021,-177.928,6.176,148.499
C04418=1205.371,170.388,-55.044,-177.924,6.177,148.498
C04419=1205.366,170.637,-55.066,-177.922,6.179,148.498
C04420=1205.362,170.886,-55.088,-177.919,6.181,148.497
C04421=1205.357,171.135,-55.109,-177.916,6.183,148.497
C04422=1205.352,171.384,-55.132,-177.914,6.184,148.497
C04423=1205.348,171.632,-55.154,-177.912,6.186,148.496
C04424=1205.343,171.882,-55.177,-177.909,6.187,148.496
C04425=1205.338,172.131,-55.199,-177.906,6.189,148.495
C04426=1205.334,172.379,-55.222,-177.903,6.191,148.495
C04427=1205.329,172.629,-55.244,-177.901,6.192,148.494
C04428=1205.325,172.877,-55.265,-177.898,6.193,148.494
C04429=1205.320,173.127,-55.288,-177.896,6.195,148.494
C04430=1205.315,173.375,-55.310,-177.893,6.197,148.493
C04431=1205.311,173.624,-55.332,-177.890,6.199,148.493
C04432=1205.306,173.874,-55.355,-177.888,6.200,148.493
C04433=1205.301,174.122,-55.377,-177.886,6.202,148.492
C04434=1205.297,174.371,-55.399,-177.883,6.203,148.492
C04435=1205.291,174.620,-55.422,-177.880,6.205,148.491
C04436=1205.287,174.869,-55.445,-177.877,6.207,148.491
C04437=1205.282,175.119,-55.467,-177.875,6.208,148.491
C04438=1205.278,175.367,-55.490,-177.872,6.210,148.490
C04439=1205.274,175.616,-55.512,-177.870,6.211,148.490
C04440=1205.268,175.865,-55.534,-177.867,6.213,148.490
C04441=1205.264,176.114,-55.557,-177.864,6.215,148.489
C04442=1205.259,176.363,-55.579,-177.862,6.216,148.489
C04443=1205.254,176.611,-55.602,-177.859,6.217,148.488
C04444=1205.250,176.861,-55.624,-177.857,6.219,148.488
C04445=1205.245,177.110,-55.647,-177.854,6.221,148.487
C04446=1205.241,177.358,-55.669,-177.851,6.223,148.487
C04447=1205.236,177.607,-55.692,-177.849,6.225,148.487
C04448=1205.232,177.857,-55.714,-177.846,6.226,148.486
C04449=1205.226,178.105,-55.737,-177.844,6.227,148.486
C04450=1205.222,178.354,-55.759,-177.841,6.229,148.486
C04451=1205.218,178.603,-55.782,-177.838,6.231,148.485
C04452=1205.212,178.852,-55.804,-177.836,6.233,148.485
C04453=1205.209,179.101,-55.827,-177.833,6.234,148.484
C04454=1205.203,179.351,-55.850,-177.831,6.235,148.484
C04455=1205.200,179.599,-55.872,-177.828,6.237,148.484
C04456=1205.194,179.848,-55.895,-177.825,6.239,148.483
C04457=1205.190,180.097,-55.917,-177.823,6.241,148.483
C04458=1205.185,180.346,-55.941,-177.820,6.243,148.483
C04459=1205.180,180.595,-55.963,-177.817,6.244,148.482
C04460=1205.176,180.844,-55.986,-177.815,6.246,148.482
C04461=1205.171,181.093,-56.009,-177.813,6.247,148.481
C04462=1205.167,181.342,-56.031,-177.810,6.249,148.481
C04463=1205.161,181.590,-56.054,-177.807,6.251,148.481
C04464=1205.157,181.839,-56.077,-177.805,6.253,148.480
C04465=1205.152,182.089,-56.100,-177.802,6.254,148.480
C04466=1205.149,182.337,-56.122,-177.799,6.256,148.480
C04467=1205.143,182.586,-56.145,-177.796,6.258,148.479
C04468=1205.139,182.835,-56.169,-177.794,6.259,148.479
C04469=1205.134,183.084,-56.191,-177.791,6.261,148.478
C04470=1205.130,183.333,-56.214,-177.789,6.262,148.478
C04471=1205.125,183.581,-56.237,-177.786,6.264,148.478
C04472=1205.120,183.830,-56.260,-177.783,6.266,148.477
C04473=1205.115,184.080,-56.283,-177.781,6.268,148.477
C04474=1205.111,184.329,-56.305,-177.778,6.270,148.477
C04475=1205.107,184.578,-56.329,-177.776,6.271,148.476
C04476=1205.102,184.847,-56.353,-177.773,6.273,148.476
C04477=1205.097,185.117,-56.378,-177.770,6.275,148.476
C04478=1205.091,185.387,-56.403,-177.767,6.277,148.475
C04479=1205.087,185.656,-56.428,-177.764,6.278,148.475
C04480=1205.082,185.905,-56.451,-177.762,6.280,148.474
C04481=1205.077,186.153,-56.474,-177.759,6.282,148.474
C04482=1205.073,186.402,-56.497,-177.756,6.284,148.474
C04483=1205.068,186.651,-56.520,-177.754,6.285,148.473
C04484=1205.063,186.900,-56.544,-177.752,6.287,148.473
C04485=1205.058,187.150,-56.566,-177.749,6.288,148.472
C04486=1205.054,187.399,-56.589,-177.746,6.290,148.472
C04487=1205.049,187.647,-56.612,-177.744,6.292,148.472
C04488=1205.044,187.896,-56.635,-177.741,6.294,148.471
C04489=1205.041,188.145,-56.658,-177.738,6.296,148.471
C04490=1205.036,188.394,-56.681,-177.736,6.297,148.471
C04491=1205.031,188.643,-56.705,-177.733,6.299,148.470
C04492=1205.026,188.892,-56.728,-177.730,6.301,148.470
C04493=1205.022,189.141,-56.751,-177.728,6.302,148.470
C04494=1205.017,189.389,-56.774,-177.726,6.304,148.469
C04495=1205.012,189.638,-56.797,-177.723,6.306,148.469
C04496=1205.008,189.887,-56.821,-177.720,6.308,148.469
C04497=1205.003,190.136,-56.844,-177.718,6.309,148.468
C04498=1204.998,190.385,-56.867,-177.715,6.311,148.468
C04499=1204.994,190.634,-56.890,-177.712,6.313,148.468
C04500=1204.990,190.883,-56.913,-177.710,6.315,148.467
C04501=1204.985,191.132,-56.937,-177.707,6.317,148.467
C04502=1204.980,191.381,-56.960,-177.704,6.318,148.466
C04503=1204.976,191.629,-56.984,-177.702,6.320,148.466
C04504=1204.971,191.877,-57.007,-177.699,6.322,148.466
C04505=1204.967,192.126,-57.030,-177.697,6.323,148.465
C04506=1204.962,192.375,-57.053,-177.694,6.325,148.465
C04507=1204.957,192.624,-57.077,-177.692,6.327,148.465
C04508=1204.953,192.873,-57.100,-177.689,6.329,148.464
C04509=1204.948,193.122,-57.123,-177.686,6.330,148.464
C04510=1204.943,193.371,-57.147,-177.684,6.332,148.464
C04511=1204.939,193.620,-57.171,-177.681,6.334,148.463
C04512=1204.934,193.869,-57.194,-177.678,6.336,148.463
C04513=1204.929,194.118,-57.218,-177.676,6.338,148.463
C04514=1204.925,194.367,-57.241,-177.673,6.339,148.462
C04515=1204.920,194.615,-57.265,-177.670,6.341,148.462
C04516=1204.916,194.864,-57.288,-177.668,6.343,148.462
C04517=1204.912,195.113,-57.311,-177.665,6.345,148.461
C04518=1204.907,195.362,-57.334,-177.662,6.347,148.461
C04519=1204.902,195.610,-57.359,-177.660,6.349,148.461
C04520=1204.898,195.860,-57.382,-177.657,6.350,148.460
C04521=1204.893,196.109,-57.405,-177.654,6.352,148.460
C04522=1204.889,196.357,-57.429,-177.652,6.353,148.459
C04523=1204.884,196.606,-57.453,-177.650,6.355,148.459
C04524=1204.879,196.855,-57.476,-177.647,6.357,148.459
C04525=1204.875,197.103,-57.500,-177.644,6.359,148.458
C04526=1204.870,197.352,-57.524,-177.642,6.360,148.458
C04527=1204.865,197.602,-57.547,-177.639,6.362,148.458
C04528=1204.861,197.850,-57.571,-177.636,6.364,148.457
C04529=1204.856,198.099,-57.594,-177.634,6.366,148.457
C04530=1204.852,198.348,-57.618,-177.631,6.368,148.457
C04531=1204.847,198.596,-57.642,-177.628,6.370,148.456
C04532=1204.842,198.846,-57.666,-177.626,6.371,148.456
C04533=1204.837,199.094,-57.690,-177.623,6.373,148.456
C04534=1204.833,199.343,-57.713,-177.621,6.375,148.455
C04535=1204.828,199.592,-57.737,-177.618,6.377,148.455
C04536=1204.824,199.841,-57.761,-177.615,6.379,148.455
C04537=1204.820,200.090,-57.784,-177.613,6.381,148.455
C04538=1204.815,200.339,-57.808,-177.610,6.383,148.454
C04539=1204.810,200.588,-57.832,-177.608,6.384,148.454
C04540=1204.806,200.836,-57.856,-177.605,6.386,148.453
C04541=1204.801,201.085,-57.879,-177.602,6.388,148.453
C04542=1204.796,201.334,-57.904,-177.600,6.390,148.453
C04543=1204.792,201.583,-57.927,-177.597,6.392,148.452
C04544=1204.787,201.831,-57.951,-177.595,6.394,148.452
C04545=1204.783,202.080,-57.975,-177.592,6.395,148.452
C04546=1204.778,202.329,-57.999,-177.589,6.397,148.451
C04547=1204.774,202.578,-58.023,-177.587,6.399,148.451
C04548=1204.770,202.827,-58.046,-177.584,6.401,148.451
C04549=1204.764,203.076,-58.071,-177.581,6.403,148.450
C04550=1204.760,203.324,-58.095,-177.579,6.405,148.450
C04551=1204.755,203.573,-58.119,-177.576,6.406,148.450
C04552=1204.751,203.822,-58.143,-177.574,6.409,148.450
C04553=1204.746,204.071,-58.166,-177.571,6.410,148.449
C04554=1204.742,204.320,-58.191,-177.569,6.412,148.449
C04555=1204.737,204.568,-58.215,-177.566,6.414,148.449
C04556=1204.733,204.818,-58.238,-177.563,6.416,148.448
C04557=1204.728,205.066,-58.263,-177.561,6.418,148.448
C04558=1204.723,205.315,-58.287,-177.558,6.419,148.448
C04559=1204.719,205.563,-58.311,-177.555,6.421,148.447
C04560=1204.715,205.813,-58.335,-177.553,6.423,148.447
C04561=1204.710,206.061,-58.359,-177.550,6.425,148.447
C04562=1204.705,206.310,-58.384,-177.547,6.427,148.446
C04563=1204.701,206.558,-58.408,-177.545,6.429,148.446
C04564=1204.696,206.807,-58.431,-177.543,6.431,148.446
C04565=1204.691,207.057,-58.456,-177.540,6.433,148.445
C04566=1204.687,207.305,-58.480,-177.537,6.434,148.445
C04567=1204.683,207.554,-58.504,-177.535,6.436,148.445
C04568=1204.678,207.802,-58.529,-177.532,6.438,148.444
C04569=1204.673,208.051,-58.552,-177.529,6.440,148.444
C04570=1204.669,208.300,-58.577,-177.527,6.442,148.444
C04571=1204.664,208.549,-58.602,-177.524,6.444,148.443
C04572=1204.660,208.798,-58.626,-177.521,6.445,148.443
C04573=1204.655,209.046,-58.650,-177.519,6.448,148.443
C04574=1204.651,209.295,-58.675,-177.517,6.449,148.443
C04575=1204.646,209.544,-58.699,-177.514,6.451,148.442
C04576=1204.641,209.793,-58.723,-177.511,6.454,148.442
C04577=1204.636,210.042,-58.747,-177.508,6.456,148.442
C04578=1204.633,210.291,-58.771,-177.505,6.458,148.441
C04579=1204.627,210.539,-58.796,-177.503,6.459,148.441
C04580=1204.622,210.810,-58.823,-177.500,6.461,148.441
C04581=1204.618,211.079,-58.849,-177.497,6.463,148.440
C04582=1204.613,211.350,-58.876,-177.494,6.466,148.440
C04583=1204.608,211.621,-58.902,-177.492,6.467,148.440
C04584=1204.603,211.870,-58.926,-177.489,6.469,148.439
C04585=1204.598,212.118,-58.951,-177.486,6.471,148.439
C04586=1204.595,212.367,-58.975,-177.484,6.473,148.439
C04587=1204.589,212.616,-59.000,-177.481,6.475,148.438
C04588=1204.585,212.865,-59.024,-177.479,6.477,148.438
C04589=1204.581,213.114,-59.049,-177.476,6.479,148.438
C04590=1204.576,213.362,-59.074,-177.474,6.481,148.437
C04591=1204.571,213.610,-59.098,-177.470,6.483,148.437
C04592=1204.567,213.860,-59.123,-177.468,6.485,148.437
C04593=1204.562,214.108,-59.147,-177.466,6.487,148.437
C04594=1204.558,214.357,-59.171,-177.463,6.489,148.436
C04595=1204.553,214.606,-59.196,-177.460,6.491,148.436
C04596=1204.549,214.855,-59.221,-177.458,6.493,148.436
C04597=1204.544,215.103,-59.245,-177.455,6.495,148.435
C04598=1204.539,215.353,-59.270,-177.452,6.496,148.435
C04599=1204.535,215.601,-59.295,-177.450,6.499,148.435
C04600=1204.530,215.849,-59.320,-177.448,6.500,148.435
C04601=1204.526,216.098,-59.344,-177.445,6.502,148.434
C04602=1204.521,216.347,-59.369,-177.442,6.504,148.434
C04603=1204.517,216.596,-59.393,-177.440,6.506,148.434
C04604=1204.513,216.844,-59.419,-177.436,6.509,148.433
C04605=1204.507,217.093,-59.443,-177.434,6.511,148.433
C04606=1204.504,217.342,-59.468,-177.432,6.513,148.433
C04607=1204.499,217.591,-59.492,-177.429,6.514,148.433
C04608=1204.495,217.839,-59.518,-177.426,6.516,148.432
C04609=1204.490,218.088,-59.542,-177.424,6.518,148.432
C04610=1204.485,218.337,-59.567,-177.421,6.520,148.432
C04611=1204.481,218.586,-59.591,-177.419,6.522,148.431
C04612=1204.476,218.834,-59.617,-177.416,6.524,148.431
C04613=1204.472,219.083,-59.642,-177.414,6.526,148.431
C04614=1204.467,219.332,-59.666,-177.410,6.528,148.430
C04615=1204.463,219.581,-59.692,-177.408,6.530,148.430
C04616=1204.458,219.829,-59.716,-177.406,6.532,148.430
C04617=1204.454,220.078,-59.740,-177.403,6.534,148.430
C04618=1204.449,220.327,-59.766,-177.400,6.536,148.429
C04619=1204.444,220.575,-59.791,-177.398,6.538,148.429
C04620=1204.440,220.824,-59.817,-177.395,6.540,148.429
C04621=1204.436,221.073,-59.841,-177.393,6.542,148.429
C04622=1204.431,221.321,-59.866,-177.390,6.544,148.428
C04623=1204.426,221.570,-59.891,-177.387,6.546,148.428
C04624=1204.422,221.819,-59.915,-177.384,6.548,148.428
C04625=1204.418,222.067,-59.941,-177.382,6.550,148.427
C04626=1204.413,222.317,-59.966,-177.380,6.552,148.427
C04627=1204.408,222.565,-59.991,-177.377,6.554,148.427
C04628=1204.404,222.814,-60.016,-177.374,6.556,148.427
C04629=1204.400,223.062,-60.041,-177.372,6.558,148.426
C04630=1204.395,223.311,-60.066,-177.370,6.560,148.426
C04631=1204.390,223.560,-60.091,-177.367,6.562,148.426
C04632=1204.386,223.809,-60.117,-177.364,6.564,148.425
C04633=1204.381,224.057,-60.142,-177.361,6.566,148.425
C04634=1204.377,224.306,-60.166,-177.358,6.568,148.425
C04635=1204.372,224.554,-60.192,-177.356,6.570,148.425
C04636=1204.368,224.803,-60.217,-177.354,6.572,148.424
C04637=1204.363,225.052,-60.242,-177.351,6.574,148.424
C04638=1204.359,225.301,-60.268,-177.348,6.576,148.424
C04639=1204.354,225.550,-60.293,-177.346,6.578,148.424
C04640=1204.350,225.798,-60.318,-177.343,6.581,148.423
C04641=1204.346,226.047,-60.343,-177.340,6.582,148.423
C04642=1204.341,226.295,-60.368,-177.338,6.584,148.423
C04643=1204.336,226.544,-60.394,-177.336,6.586,148.423
C04644=1204.332,226.792,-60.419,-177.333,6.588,148.422
C04645=1204.327,227.042,-60.444,-177.330,6.590,148.422
C04646=1204.323,227.291,-60.470,-177.328,6.592,148.422
C04647=1204.318,227.539,-60.495,-177.325,6.595,148.422
C04648=1204.314,227.787,-60.521,-177.322,6.597,148.421
C04649=1204.309,228.036,-60.546,-177.320,6.599,148.421
C04650=1204.304,228.285,-60.572,-177.317,6.601,148.421
C04651=1204.300,228.534,-60.597,-177.315,6.603,148.420
C04652=1204.295,228.782,-60.622,-177.312,6.605,148.420
C04653=1204.292,229.031,-60.647,-177.310,6.606,148.420
C04654=1204.287,229.279,-60.673,-177.307,6.609,148.420
C04655=1204.283,229.528,-60.698,-177.304,6.611,148.419
C04656=1204.278,229.777,-60.724,-177.302,6.613,148.419
C04657=1204.273,230.025,-60.749,-177.299,6.615,148.419
C04658=1204.269,230.274,-60.775,-177.297,6.617,148.419
C04659=1204.265,230.523,-60.800,-177.294,6.619,148.418
C04660=1204.260,230.771,-60.826,-177.291,6.622,148.418
C04661=1204.256,231.020,-60.851,-177.289,6.624,148.418
C04662=1204.250,231.268,-60.877,-177.286,6.626,148.418
C04663=1204.246,231.517,-60.903,-177.284,6.627,148.417
C04664=1204.242,231.766,-60.929,-177.281,6.630,148.417
C04665=1204.237,232.015,-60.954,-177.279,6.631,148.417
C04666=1204.232,232.263,-60.979,-177.276,6.634,148.417
C04667=1204.228,232.512,-61.005,-177.273,6.636,148.416
C04668=1204.224,232.761,-61.031,-177.271,6.638,148.416
C04669=1204.219,233.009,-61.056,-177.268,6.640,148.416
C04670=1204.215,233.258,-61.082,-177.265,6.642,148.416
C04671=1204.211,233.507,-61.108,-177.263,6.644,148.415
C04672=1204.206,233.755,-61.133,-177.260,6.647,148.415
C04673=1204.202,234.004,-61.159,-177.257,6.648,148.415
C04674=1204.197,234.253,-61.185,-177.255,6.651,148.415
C04675=1204.192,234.501,-61.211,-177.253,6.652,148.414
C04676=1204.188,234.750,-61.236,-177.250,6.654,148.414
C04677=1204.183,234.999,-61.262,-177.248,6.656,148.414
C04678=1204.179,235.247,-61.288,-177.245,6.659,148.414
C04679=1204.174,235.495,-61.313,-177.242,6.661,148.413
C04680=1204.170,235.744,-61.340,-177.240,6.663,148.413
C04681=1204.165,235.993,-61.366,-177.237,6.665,148.413
C04682=1204.161,236.242,-61.392,-177.235,6.667,148.413
C04683=1204.156,236.490,-61.417,-177.232,6.670,148.413
C04684=1204.152,236.762,-61.445,-177.229,6.672,148.412
C04685=1204.147,237.033,-61.474,-177.226,6.674,148.412
C04686=1204.142,237.304,-61.502,-177.224,6.676,148.412
C04687=1204.137,237.576,-61.530,-177.220,6.679,148.411
C04688=1204.133,237.824,-61.557,-177.218,6.681,148.411
C04689=1204.128,238.073,-61.582,-177.216,6.683,148.411
C04690=1204.124,238.321,-61.608,-177.213,6.685,148.411
C04691=1204.119,238.570,-61.634,-177.211,6.687,148.411
C04692=1204.114,238.819,-61.660,-177.208,6.690,148.410
C04693=1204.110,239.067,-61.686,-177.205,6.692,148.410
C04694=1204.106,239.316,-61.712,-177.203,6.694,148.410
C04695=1204.101,239.565,-61.738,-177.200,6.695,148.409
C04696=1204.096,239.813,-61.764,-177.198,6.698,148.409
C04697=1204.093,240.062,-61.790,-177.195,6.700,148.409
C04698=1204.088,240.311,-61.817,-177.192,6.702,148.409
C04699=1204.083,240.560,-61.842,-177.190,6.704,148.409
C04700=1204.079,240.807,-61.869,-177.187,6.706,148.408
C04701=1204.074,241.056,-61.895,-177.185,6.709,148.408
C04702=1204.070,241.305,-61.921,-177.182,6.711,148.408
C04703=1204.066,241.553,-61.947,-177.179,6.713,148.408
C04704=1204.061,241.802,-61.973,-177.177,6.715,148.408
C04705=1204.057,242.051,-61.999,-177.175,6.717,148.407
C04706=1204.053,242.299,-62.026,-177.172,6.720,148.407
C04707=1204.047,242.548,-62.052,-177.169,6.722,148.407
C04708=1204.043,242.796,-62.078,-177.167,6.724,148.407
C04709=1204.038,243.045,-62.104,-177.165,6.726,148.406
C04710=1204.034,243.294,-62.130,-177.161,6.728,148.406
C04711=1204.030,243.542,-62.157,-177.159,6.731,148.406
C04712=1204.025,243.791,-62.183,-177.157,6.732,148.406
C04713=1204.021,244.039,-62.210,-177.154,6.734,148.405
C04714=1204.016,244.288,-62.236,-177.151,6.737,148.405
C04715=1204.012,244.537,-62.262,-177.149,6.739,148.405
C04716=1204.007,244.785,-62.288,-177.146,6.741,148.405
C04717=1204.003,245.033,-62.315,-177.144,6.743,148.405
C04718=1203.999,245.282,-62.341,-177.141,6.746,148.404
C04719=1203.994,245.530,-62.368,-177.138,6.748,148.404
C04720=1203.990,245.779,-62.393,-177.136,6.750,148.404
C04721=1203.985,246.028,-62.420,-177.134,6.752,148.404
C04722=1203.981,246.276,-62.447,-177.130,6.755,148.404
C04723=1203.976,246.525,-62.473,-177.128,6.757,148.404
C04724=1203.972,246.773,-62.500,-177.126,6.759,148.403
C04725=1203.967,247.022,-62.526,-177.123,6.761,148.403
C04726=1203.963,247.271,-62.552,-177.120,6.764,148.403
C04727=1203.959,247.519,-62.580,-177.118,6.765,148.403
C04728=1203.954,247.768,-62.605,-177.116,6.768,148.402
C04729=1203.950,248.016,-62.632,-177.113,6.769,148.402
C04730=1203.945,248.265,-62.659,-177.110,6.772,148.402
C04731=1203.941,248.514,-62.685,-177.108,6.774,148.402
C04732=1203.936,248.762,-62.712,-177.105,6.777,148.402
C04733=1203.932,249.010,-62.739,-177.103,6.778,148.401
C04734=1203.927,249.259,-62.765,-177.100,6.781,148.401
C04735=1203.923,249.508,-62.792,-177.098,6.783,148.401
C04736=1203.919,249.756,-62.819,-177.095,6.785,148.401
C04737=1203.914,250.005,-62.846,-177.092,6.788,148.401
C04738=1203.910,250.253,-62.871,-177.090,6.790,148.400
C04739=1203.905,250.502,-62.898,-177.087,6.792,148.400
C04740=1203.901,250.750,-62.926,-177.085,6.794,148.400
C04741=1203.897,250.999,-62.952,-177.082,6.797,148.400
C04742=1203.892,251.248,-62.978,-177.079,6.799,148.400
C04743=1203.887,251.496,-63.005,-177.077,6.801,148.399
C04744=1203.883,251.744,-63.032,-177.074,6.804,148.399
C04745=1203.879,251.993,-63.059,-177.072,6.806,148.399
C04746=1203.874,252.241,-63.086,-177.069,6.808,148.399
C04747=1203.870,252.490,-63.112,-177.067,6.811,148.399
C04748=1203.865,252.738,-63.139,-177.064,6.813,148.398
C04749=1203.860,252.987,-63.166,-177.061,6.814,148.398
C04750=1203.856,253.235,-63.192,-177.059,6.817,148.398
C04751=1203.852,253.484,-63.219,-177.056,6.819,148.398
C04752=1203.847,253.732,-63.246,-177.054,6.821,148.398
C04753=1203.843,253.981,-63.273,-177.051,6.823,148.397
C04754=1203.839,254.230,-63.300,-177.049,6.826,148.397
C04755=1203.834,254.478,-63.327,-177.046,6.828,148.397
C04756=1203.830,254.727,-63.354,-177.044,6.830,148.397
C04757=1203.826,254.975,-63.381,-177.041,6.833,148.397
C04758=1203.821,255.223,-63.408,-177.038,6.835,148.397
C04759=1203.817,255.472,-63.435,-177.036,6.837,148.396
C04760=1203.812,255.720,-63.462,-177.033,6.840,148.396
C04761=1203.807,255.969,-63.489,-177.031,6.842,148.396
C04762=1203.803,256.217,-63.516,-177.028,6.844,148.396
C04763=1203.799,256.466,-63.543,-177.026,6.847,148.396
C04764=1203.795,256.715,-63.570,-177.023,6.849,148.395
C04765=1203.790,256.963,-63.597,-177.021,6.851,148.395
C04766=1203.785,257.212,-63.624,-177.018,6.854,148.395
C04767=1203.781,257.460,-63.651,-177.016,6.856,148.395
C04768=1203.777,257.708,-63.678,-177.013,6.858,148.395
C04769=1203.772,257.956,-63.706,-177.010,6.861,148.395
C04770=1203.768,258.206,-63.733,-177.008,6.863,148.394
C04771=1203.764,258.454,-63.760,-177.005,6.865,148.394
C04772=1203.759,258.703,-63.787,-177.002,6.868,148.394
C04773=1203.754,258.951,-63.814,-177.000,6.870,148.394
C04774=1203.750,259.199,-63.841,-176.998,6.872,148.394
C04775=1203.745,259.447,-63.869,-176.995,6.875,148.394
C04776=1203.742,259.696,-63.896,-176.992,6.876,148.393
C04777=1203.737,259.945,-63.923,-176.990,6.879,148.393
C04778=1203.733,260.193,-63.950,-176.987,6.882,148.393
C04779=1203.728,260.441,-63.978,-176.985,6.884,148.393
C04780=1203.724,260.690,-64.005,-176.983,6.886,148.393
C04781=1203.720,260.939,-64.032,-176.979,6.888,148.392
C04782=1203.715,261.187,-64.059,-176.977,6.891,148.392
C04783=1203.711,261.435,-64.087,-176.975,6.892,148.392
C04784=1203.706,261.684,-64.114,-176.972,6.895,148.392
C04785=1203.702,261.933,-64.142,-176.970,6.898,148.392
C04786=1203.698,262.181,-64.169,-176.967,6.900,148.392
C04787=1203.693,262.429,-64.196,-176.964,6.902,148.392
C04788=1203.688,262.702,-64.227,-176.961,6.905,148.391
C04789=1203.684,262.975,-64.257,-176.959,6.907,148.391
C04790=1203.678,263.248,-64.287,-176.956,6.910,148.391
C04791=1203.674,263.520,-64.317,-176.953,6.913,148.391
C04792=1203.670,263.769,-64.344,-176.951,6.915,148.391
C04793=1203.665,264.018,-64.372,-176.948,6.917,148.391
C04794=1203.660,264.266,-64.400,-176.945,6.920,148.390
C04795=1203.656,264.514,-64.427,-176.943,6.922,148.390
C04796=1203.652,264.763,-64.455,-176.940,6.925,148.390
C04797=1203.647,265.011,-64.482,-176.938,6.927,148.390
C04798=1203.643,265.259,-64.510,-176.936,6.929,148.390
C04799=1203.639,265.508,-64.537,-176.933,6.932,148.390
C04800=1203.634,265.756,-64.565,-176.930,6.934,148.389
C04801=1203.630,266.005,-64.592,-176.927,6.937,148.389
C04802=1203.625,266.253,-64.620,-176.925,6.939,148.389
C04803=1203.621,266.502,-64.647,-176.923,6.941,148.389
C04804=1203.616,266.750,-64.676,-176.920,6.944,148.389
C04805=1203.612,266.998,-64.703,-176.918,6.946,148.389
C04806=1203.608,267.247,-64.731,-176.914,6.949,148.388
C04807=1203.603,267.496,-64.758,-176.912,6.951,148.388
C04808=1203.599,267.743,-64.786,-176.910,6.953,148.388
C04809=1203.595,267.992,-64.814,-176.907,6.956,148.388
C04810=1203.590,268.241,-64.841,-176.905,6.958,148.388
C04811=1203.586,268.489,-64.870,-176.902,6.961,148.388
C04812=1203.581,268.738,-64.897,-176.900,6.963,148.388
C04813=1203.577,268.986,-64.924,-176.897,6.965,148.388
C04814=1203.573,269.234,-64.953,-176.895,6.968,148.387
C04815=1203.568,269.483,-64.980,-176.892,6.970,148.387
C04816=1203.563,269.731,-65.008,-176.889,6.973,148.387
C04817=1203.560,269.980,-65.036,-176.887,6.975,148.387
C04818=1203.555,270.227,-65.064,-176.885,6.977,148.387
C04819=1203.550,270.477,-65.092,-176.882,6.980,148.387
C04820=1203.546,270.725,-65.120,-176.879,6.982,148.386
C04821=1203.542,270.973,-65.147,-176.877,6.985,148.386
C04822=1203.538,271.221,-65.176,-176.874,6.987,148.386
C04823=1203.533,271.470,-65.203,-176.871,6.990,148.386
C04824=1203.529,271.719,-65.231,-176.869,6.992,148.386
C04825=1203.525,271.967,-65.259,-176.866,6.995,148.386
C04826=1203.519,272.215,-65.288,-176.864,6.997,148.386
C04827=1203.515,272.464,-65.315,-176.862,6.999,148.386
C04828=1203.511,272.712,-65.343,-176.859,7.002,148.386
C04829=1203.507,272.961,-65.371,-176.856,7.004,148.385
C04830=1203.502,273.209,-65.399,-176.854,7.007,148.385
C04831=1203.498,273.457,-65.427,-176.851,7.009,148.385
C04832=1203.493,273.705,-65.456,-176.848,7.012,148.385
C04833=1203.490,273.954,-65.484,-176.846,7.014,148.385
C04834=1203.485,274.202,-65.512,-176.844,7.016,148.385
C04835=1203.480,274.451,-65.540,-176.841,7.019,148.385
C04836=1203.476,274.699,-65.567,-176.839,7.021,148.384
C04837=1203.472,274.948,-65.596,-176.836,7.024,148.384
C04838=1203.467,275.196,-65.624,-176.834,7.026,148.384
C04839=1203.464,275.445,-65.652,-176.831,7.029,148.384
C04840=1203.458,275.693,-65.681,-176.829,7.031,148.384
C04841=1203.455,275.941,-65.709,-176.826,7.034,148.384
C04842=1203.450,276.189,-65.736,-176.823,7.036,148.384
C04843=1203.446,276.438,-65.765,-176.821,7.039,148.384
C04844=1203.442,276.686,-65.793,-176.818,7.041,148.384
C04845=1203.437,276.935,-65.822,-176.816,7.044,148.383
C04846=1203.433,277.183,-65.849,-176.813,7.046,148.383
C04847=1203.428,277.432,-65.878,-176.811,7.048,148.383
C04848=1203.424,277.679,-65.906,-176.808,7.051,148.383
C04849=1203.420,277.928,-65.935,-176.806,7.053,148.383
C04850=1203.415,278.176,-65.963,-176.803,7.056,148.383
C04851=1203.411,278.424,-65.992,-176.801,7.058,148.383
C04852=1203.406,278.672,-66.020,-176.798,7.061,148.383
C04853=1203.402,278.921,-66.048,-176.796,7.063,148.382
C04854=1203.398,279.170,-66.077,-176.793,7.066,148.382
C04855=1203.393,279.418,-66.105,-176.791,7.068,148.382
C04856=1203.390,279.666,-66.134,-176.788,7.071,148.382
C04857=1203.385,279.914,-66.162,-176.785,7.073,148.382
C04858=1203.381,280.163,-66.190,-176.783,7.076,148.382
C04859=1203.376,280.411,-66.219,-176.781,7.078,148.382
C04860=1203.372,280.659,-66.247,-176.778,7.081,148.382
C04861=1203.368,280.908,-66.276,-176.775,7.083,148.382
C04862=1203.363,281.156,-66.305,-176.773,7.086,148.381
C04863=1203.359,281.405,-66.333,-176.770,7.088,148.381
C04864=1203.355,281.653,-66.362,-176.768,7.091,148.381
C04865=1203.350,281.901,-66.390,-176.765,7.093,148.381
C04866=1203.346,282.150,-66.419,-176.762,7.096,148.381
C04867=1203.341,282.398,-66.447,-176.760,7.098,148.381
C04868=1203.337,282.646,-66.476,-176.758,7.101,148.381
C04869=1203.333,282.895,-66.505,-176.755,7.104,148.381
C04870=1203.328,283.143,-66.533,-176.752,7.106,148.381
C04871=1203.324,283.391,-66.562,-176.750,7.108,148.381
C04872=1203.320,283.640,-66.591,-176.747,7.112,148.381
C04873=1203.315,283.888,-66.619,-176.745,7.114,148.380
C04874=1203.311,284.136,-66.648,-176.743,7.117,148.380
C04875=1203.307,284.385,-66.677,-176.740,7.119,148.380
C04876=1203.302,284.633,-66.705,-176.737,7.122,148.380
C04877=1203.298,284.881,-66.734,-176.735,7.124,148.380
C04878=1203.294,285.130,-66.763,-176.732,7.127,148.380
C04879=1203.289,285.377,-66.792,-176.730,7.129,148.380
C04880=1203.285,285.626,-66.821,-176.727,7.132,148.380
C04881=1203.281,285.874,-66.849,-176.725,7.134,148.380
C04882=1203.276,286.122,-66.878,-176.722,7.137,148.380
C04883=1203.272,286.371,-66.907,-176.720,7.139,148.380
C04884=1203.267,286.619,-66.936,-176.717,7.142,148.380
C04885=1203.263,286.867,-66.964,-176.714,7.145,148.379
C04886=1203.259,287.116,-66.993,-176.712,7.147,148.379
C04887=1203.255,287.364,-67.023,-176.709,7.150,148.379
C04888=1203.250,287.613,-67.051,-176.707,7.152,148.379
C04889=1203.245,287.860,-67.080,-176.705,7.155,148.379
C04890=1203.242,288.108,-67.109,-176.702,7.157,148.379
C04891=1203.238,288.357,-67.138,-176.699,7.160,148.379
C04892=1203.233,288.631,-67.170,-176.697,7.163,148.379
C04893=1203.227,288.906,-67.203,-176.694,7.166,148.379
C04894=1203.223,289.180,-67.234,-176.692,7.168,148.379
C04895=1203.218,289.454,-67.266,-176.689,7.171,148.378
C04896=1203.214,289.703,-67.295,-176.686,7.174,148.378
C04897=1203.209,289.951,-67.325,-176.684,7.176,148.378
C04898=1203.205,290.200,-67.354,-176.681,7.179,148.378
C04899=1203.201,290.448,-67.383,-176.678,7.182,148.378
C04900=1203.196,290.696,-67.412,-176.676,7.184,148.378
C04901=1203.193,290.943,-67.441,-176.674,7.187,148.378
C04902=1203.188,291.192,-67.470,-176.671,7.190,148.378
C04903=1203.184,291.441,-67.499,-176.668,7.192,148.378
C04904=1203.180,291.689,-67.529,-176.666,7.195,148.378
C04905=1203.175,291.936,-67.558,-176.663,7.198,148.378
C04906=1203.170,292.185,-67.586,-176.661,7.200,148.378
C04907=1203.166,292.434,-67.616,-176.659,7.203,148.378
C04908=1203.162,292.682,-67.645,-176.656,7.206,148.378
C04909=1203.158,292.930,-67.675,-176.654,7.208,148.378
C04910=1203.153,293.178,-67.704,-176.651,7.211,148.378
C04911=1203.149,293.426,-67.733,-176.649,7.213,148.378
C04912=1203.144,293.675,-67.762,-176.646,7.216,148.377
C04913=1203.140,293.923,-67.792,-176.644,7.218,148.377
C04914=1203.136,294.171,-67.821,-176.641,7.221,148.377
C04915=1203.132,294.420,-67.850,-176.638,7.224,148.377
C04916=1203.128,294.668,-67.880,-176.636,7.226,148.377
C04917=1203.123,294.915,-67.909,-176.633,7.229,148.377
C04918=1203.119,295.164,-67.938,-176.631,7.232,148.377
C04919=1203.115,295.412,-67.968,-176.629,7.235,148.377
C04920=1203.110,295.660,-67.997,-176.627,7.237,148.377
C04921=1203.106,295.909,-68.027,-176.624,7.240,148.377
C04922=1203.102,296.157,-68.056,-176.621,7.243,148.377
C04923=1203.098,296.405,-68.086,-176.619,7.245,148.377
C04924=1203.094,296.653,-68.115,-176.616,7.248,148.377
C04925=1203.090,296.902,-68.145,-176.614,7.250,148.377
C04926=1203.085,297.150,-68.174,-176.611,7.253,148.377
C04927=1203.080,297.398,-68.204,-176.609,7.256,148.377
C04928=1203.076,297.646,-68.233,-176.607,7.258,148.377
C04929=1203.071,297.894,-68.263,-176.603,7.261,148.376
C04930=1203.067,298.143,-68.292,-176.601,7.263,148.376
C04931=1203.063,298.391,-68.322,-176.599,7.266,148.376
C04932=1203.059,298.639,-68.351,-176.597,7.269,148.376
C04933=1203.055,298.887,-68.380,-176.594,7.272,148.376
C04934=1203.051,299.136,-68.410,-176.591,7.275,148.376
C04935=1203.046,299.384,-68.441,-176.589,7.277,148.376
C04936=1203.042,299.632,-68.470,-176.586,7.280,148.376
C04937=1203.038,299.880,-68.500,-176.584,7.282,148.376
C04938=1203.033,300.128,-68.529,-176.581,7.285,148.376
C04939=1203.029,300.377,-68.558,-176.579,7.288,148.376
C04940=1203.024,300.625,-68.589,-176.577,7.290,148.376
C04941=1203.020,300.873,-68.619,-176.574,7.293,148.376
C04942=1203.016,301.121,-68.648,-176.572,7.295,148.376
C04943=1203.012,301.369,-68.678,-176.569,7.298,148.376
C04944=1203.007,301.618,-68.708,-176.566,7.302,148.376
C04945=1203.003,301.866,-68.738,-176.564,7.304,148.376
C04946=1202.999,302.114,-68.767,-176.562,7.307,148.376
C04947=1202.995,302.362,-68.797,-176.560,7.309,148.376
C04948=1202.990,302.610,-68.827,-176.557,7.312,148.376
C04949=1202.986,302.858,-68.857,-176.555,7.315,148.376
C04950=1202.982,303.107,-68.886,-176.552,7.317,148.376
C04951=1202.977,303.355,-68.917,-176.550,7.320,148.376
C04952=1202.973,303.603,-68.947,-176.547,7.324,148.376
C04953=1202.969,303.851,-68.976,-176.545,7.326,148.376
C04954=1202.965,304.099,-69.006,-176.542,7.329,148.376
C04955=1202.960,304.347,-69.036,-176.540,7.331,148.376
C04956=1202.956,304.596,-69.066,-176.537,7.334,148.376
C04957=1202.951,304.844,-69.096,-176.535,7.337,148.376
C04958=1202.947,305.092,-69.126,-176.533,7.339,148.376
C04959=1202.943,305.340,-69.156,-176.530,7.342,148.376
C04960=1202.938,305.588,-69.186,-176.527,7.345,148.376
C04961=1202.934,305.836,-69.216,-176.525,7.347,148.376
C04962=1202.931,306.085,-69.246,-176.522,7.350,148.376
C04963=1202.926,306.333,-69.277,-176.521,7.353,148.376
C04964=1202.922,306.581,-69.306,-176.518,7.356,148.376
C04965=1202.918,306.829,-69.337,-176.515,7.359,148.376
C04966=1202.913,307.077,-69.367,-176.513,7.361,148.376
C04967=1202.909,307.325,-69.397,-176.511,7.364,148.376
C04968=1202.905,307.573,-69.427,-176.508,7.367,148.376
C04969=1202.901,307.821,-69.457,-176.506,7.369,148.376
C04970=1202.896,308.070,-69.487,-176.503,7.372,148.376
C04971=1202.892,308.317,-69.517,-176.501,7.375,148.375
C04972=1202.888,308.567,-69.548,-176.499,7.378,148.376
C04973=1202.884,308.814,-69.578,-176.496,7.381,148.376
C04974=1202.879,309.062,-69.609,-176.494,7.383,148.376
C04975=1202.875,309.310,-69.638,-176.491,7.386,148.376
C04976=1202.870,309.558,-69.669,-176.488,7.389,148.376
C04977=1202.866,309.806,-69.699,-176.486,7.391,148.376
C04978=1202.861,310.055,-69.729,-176.484,7.394,148.376
C04979=1202.858,310.303,-69.760,-176.481,7.398,148.376
C04980=1202.854,310.551,-69.790,-176.479,7.400,148.376
C04981=1202.849,310.799,-69.820,-176.477,7.403,148.376
C04982=1202.845,311.047,-69.850,-176.475,7.405,148.376
C04983=1202.841,311.295,-69.881,-176.472,7.408,148.376
C04984=1202.837,311.543,-69.912,-176.469,7.411,148.376
C04985=1202.832,311.792,-69.942,-176.467,7.414,148.376
C04986=1202.828,312.040,-69.972,-176.465,7.417,148.376
C04987=1202.823,312.288,-70.003,-176.462,7.420,148.376
C04988=1202.820,312.535,-70.033,-176.460,7.422,148.376
C04989=1202.816,312.784,-70.064,-176.457,7.425,148.376
C04990=1202.811,313.033,-70.094,-176.455,7.428,148.376
C04991=1202.807,313.280,-70.124,-176.453,7.431,148.376
C04992=1202.802,313.528,-70.155,-176.450,7.434,148.376
C04993=1202.798,313.776,-70.185,-176.448,7.437,148.376
C04994=1202.794,314.024,-70.216,-176.445,7.439,148.376
C04995=1202.790,314.272,-70.247,-176.443,7.442,148.376
C04996=1202.785,314.549,-70.281,-176.441,7.445,148.376
C04997=1202.780,314.825,-70.315,-176.438,7.448,148.376
C04998=1202.775,315.102,-70.349,-176.435,7.451,148.376
C04999=1202.771,315.378,-70.383,-176.432,7.454,148.376
C05000=1202.767,315.625,-70.413,-176.430,7.457,148.376
C05001=1202.762,315.873,-70.444,-176.428,7.461,148.376
C05002=1202.758,316.122,-70.475,-176.425,7.463,148.376
C05003=1202.754,316.369,-70.505,-176.423,7.466,148.376
C05004=1202.750,316.617,-70.536,-176.421,7.469,148.376
C05005=1202.746,316.866,-70.567,-176.418,7.471,148.376
C05006=1202.741,317.114,-70.598,-176.416,7.474,148.376
C05007=1202.737,317.362,-70.628,-176.414,7.477,148.376
C05008=1202.733,317.610,-70.659,-176.411,7.480,148.376
C05009=1202.728,317.858,-70.690,-176.409,7.483,148.376
C05010=1202.724,318.106,-70.721,-176.407,7.485,148.376
C05011=1202.720,318.354,-70.751,-176.404,7.489,148.377
C05012=1202.716,318.603,-70.782,-176.402,7.492,148.377
C05013=1202.711,318.850,-70.813,-176.399,7.494,148.377
C05014=1202.707,319.098,-70.844,-176.397,7.497,148.377
C05015=1202.703,319.346,-70.876,-176.395,7.500,148.377
C05016=1202.699,319.594,-70.906,-176.392,7.502,148.377
C05017=1202.695,319.843,-70.937,-176.390,7.505,148.377
C05018=1202.691,320.091,-70.968,-176.388,7.509,148.377
C05019=1202.686,320.339,-70.998,-176.385,7.511,148.377
C05020=1202.682,320.587,-71.030,-176.383,7.514,148.377
C05021=1202.678,320.835,-71.061,-176.381,7.517,148.377
C05022=1202.674,321.082,-71.091,-176.378,7.519,148.377
C05023=1202.670,321.331,-71.122,-176.376,7.523,148.377
C05024=1202.665,321.578,-71.154,-176.373,7.526,148.377
C05025=1202.661,321.826,-71.185,-176.371,7.528,148.377
C05026=1202.657,322.075,-71.216,-176.369,7.531,148.377
C05027=1202.652,322.323,-71.246,-176.366,7.534,148.377
C05028=1202.648,322.571,-71.278,-176.364,7.537,148.377
C05029=1202.644,322.819,-71.309,-176.362,7.540,148.378
C05030=1202.640,323.068,-71.340,-176.359,7.543,148.378
C05031=1202.636,323.315,-71.372,-176.357,7.546,148.378
C05032=1202.632,323.563,-71.402,-176.355,7.548,148.378
C05033=1202.628,323.811,-71.433,-176.352,7.551,148.378
C05034=1202.623,324.059,-71.464,-176.350,7.555,148.378
C05035=1202.619,324.307,-71.496,-176.348,7.557,148.378
C05036=1202.615,324.555,-71.526,-176.346,7.560,148.378
C05037=1202.611,324.803,-71.558,-176.343,7.563,148.378
C05038=1202.606,325.051,-71.589,-176.341,7.566,148.378
C05039=1202.602,325.299,-71.620,-176.339,7.569,148.378
C05040=1202.598,325.547,-71.652,-176.336,7.572,148.378
C05041=1202.594,325.795,-71.683,-176.334,7.574,148.378
C05042=1202.590,326.043,-71.714,-176.332,7.577,148.378
C05043=1202.585,326.291,-71.746,-176.330,7.581,148.379
C05044=1202.581,326.539,-71.777,-176.327,7.583,148.379
C05045=1202.577,326.786,-71.808,-176.325,7.586,148.379
C05046=1202.573,327.035,-71.839,-176.322,7.589,148.379
C05047=1202.569,327.282,-71.871,-176.321,7.592,148.379
C05048=1202.565,327.531,-71.902,-176.318,7.595,148.379
C05049=1202.560,327.779,-71.934,-176.316,7.598,148.379
C05050=1202.556,328.027,-71.965,-176.314,7.600,148.379
C05051=1202.551,328.275,-71.997,-176.312,7.604,148.379
C05052=1202.547,328.523,-72.028,-176.309,7.607,148.379
C05053=1202.543,328.771,-72.059,-176.307,7.609,148.379
C05054=1202.539,329.019,-72.091,-176.305,7.612,148.379
C05055=1202.535,329.267,-72.122,-176.302,7.616,148.380
C05056=1202.531,329.515,-72.154,-176.300,7.618,148.380
C05057=1202.527,329.762,-72.185,-176.298,7.621,148.380
C05058=1202.522,330.011,-72.217,-176.296,7.625,148.380
C05059=1202.518,330.259,-72.249,-176.293,7.628,148.380
C05060=1202.514,330.507,-72.280,-176.291,7.630,148.380
C05061=1202.510,330.755,-72.311,-176.289,7.633,148.380
C05062=1202.506,331.003,-72.343,-176.287,7.636,148.380
C05063=1202.502,331.251,-72.375,-176.284,7.639,148.380
C05064=1202.497,331.499,-72.406,-176.282,7.642,148.381
C05065=1202.493,331.747,-72.438,-176.280,7.645,148.381
C05066=1202.489,331.994,-72.469,-176.278,7.648,148.381
C05067=1202.485,332.242,-72.501,-176.276,7.651,148.381
C05068=1202.480,332.491,-72.534,-176.273,7.654,148.381
C05069=1202.476,332.739,-72.564,-176.271,7.656,148.381
C05070=1202.472,332.987,-72.596,-176.269,7.660,148.381
C05071=1202.468,333.234,-72.628,-176.266,7.663,148.381
C05072=1202.464,333.482,-72.660,-176.265,7.665,148.382
C05073=1202.460,333.730,-72.692,-176.262,7.669,148.382
C05074=1202.455,333.978,-72.724,-176.260,7.672,148.382
C05075=1202.451,334.226,-72.755,-176.258,7.674,148.382
C05076=1202.446,334.474,-72.787,-176.255,7.677,148.382
C05077=1202.443,334.722,-72.819,-176.253,7.681,148.382
C05078=1202.439,334.970,-72.850,-176.252,7.683,148.382
C05079=1202.435,335.217,-72.882,-176.249,7.686,148.383
C05080=1202.430,335.466,-72.914,-176.247,7.689,148.383
C05081=1202.426,335.714,-72.946,-176.245,7.692,148.383
C05082=1202.422,335.961,-72.978,-176.243,7.695,148.383
C05083=1202.418,336.209,-73.010,-176.240,7.698,148.383
C05084=1202.414,336.457,-73.042,-176.238,7.702,148.383
C05085=1202.410,336.705,-73.073,-176.236,7.704,148.383
C05086=1202.405,336.953,-73.106,-176.234,7.707,148.383
C05087=1202.402,337.201,-73.138,-176.231,7.711,148.384
C05088=1202.396,337.449,-73.170,-176.230,7.713,148.384
C05089=1202.393,337.697,-73.202,-176.227,7.716,148.384
C05090=1202.389,337.945,-73.233,-176.225,7.719,148.384
C05091=1202.384,338.193,-73.266,-176.223,7.722,148.384
C05092=1202.380,338.441,-73.297,-176.221,7.725,148.384
C05093=1202.376,338.689,-73.330,-176.219,7.729,148.385
C05094=1202.372,338.937,-73.362,-176.217,7.731,148.385
C05095=1202.368,339.184,-73.393,-176.214,7.734,148.385
C05096=1202.363,339.433,-73.426,-176.212,7.737,148.385
C05097=1202.360,339.680,-73.458,-176.210,7.740,148.385
C05098=1202.355,339.928,-73.490,-176.208,7.743,148.385
C05099=1202.351,340.176,-73.522,-176.206,7.747,148.386
C05100=1202.347,340.454,-73.559,-176.203,7.750,148.386
C05101=1202.341,340.733,-73.594,-176.201,7.753,148.386
C05102=1202.337,341.011,-73.631,-176.199,7.756,148.386
C05103=1202.332,341.289,-73.667,-176.197,7.760,148.386
C05104=1202.328,341.537,-73.699,-176.194,7.763,148.387
C05105=1202.324,341.786,-73.731,-176.192,7.766,148.387
C05106=1202.320,342.033,-73.764,-176.190,7.769,148.387
C05107=1202.315,342.281,-73.796,-176.188,7.772,148.387
C05108=1202.312,342.529,-73.828,-176.186,7.775,148.387
C05109=1202.307,342.777,-73.860,-176.184,7.778,148.387
C05110=1202.304,343.024,-73.893,-176.182,7.781,148.388
C05111=1202.299,343.272,-73.925,-176.179,7.784,148.388
C05112=1202.295,343.520,-73.957,-176.178,7.787,148.388
C05113=1202.291,343.768,-73.990,-176.176,7.790,148.388
C05114=1202.286,344.016,-74.022,-176.173,7.794,148.388
C05115=1202.283,344.264,-74.054,-176.172,7.796,148.389
C05116=1202.278,344.511,-74.087,-176.169,7.799,148.389
C05117=1202.274,344.759,-74.119,-176.167,7.802,148.389
C05118=1202.270,345.008,-74.151,-176.165,7.805,148.389
C05119=1202.266,345.255,-74.184,-176.163,7.808,148.389
C05120=1202.262,345.503,-74.216,-176.161,7.812,148.389
C05121=1202.257,345.751,-74.249,-176.159,7.814,148.390
C05122=1202.253,345.999,-74.281,-176.157,7.818,148.390
C05123=1202.249,346.246,-74.314,-176.155,7.821,148.390
C05124=1202.245,346.495,-74.346,-176.153,7.823,148.390
C05125=1202.241,346.742,-74.379,-176.151,7.827,148.391
C05126=1202.237,346.990,-74.411,-176.148,7.830,148.391
C05127=1202.232,347.238,-74.443,-176.147,7.833,148.391
C05128=1202.228,347.486,-74.477,-176.145,7.836,148.391
C05129=1202.225,347.733,-74.509,-176.143,7.839,148.392
C05130=1202.220,347.982,-74.542,-176.141,7.842,148.392
C05131=1202.216,348.229,-74.575,-176.139,7.845,148.392
C05132=1202.212,348.477,-74.607,-176.137,7.848,148.392
C05133=1202.208,348.725,-74.640,-176.135,7.851,148.392
C05134=1202.203,348.973,-74.672,-176.133,7.855,148.393
C05135=1202.199,349.220,-74.705,-176.131,7.857,148.393
C05136=1202.195,349.468,-74.737,-176.129,7.860,148.393
C05137=1202.191,349.716,-74.770,-176.127,7.864,148.393
C05138=1202.187,349.964,-74.803,-176.125,7.866,148.393
C05139=1202.183,350.212,-74.836,-176.123,7.870,148.394
C05140=1202.179,350.460,-74.868,-176.121,7.873,148.394
C05141=1202.175,350.707,-74.901,-176.119,7.876,148.394
C05142=1202.171,350.956,-74.934,-176.117,7.879,148.394
C05143=1202.166,351.204,-74.967,-176.115,7.882,148.395
C05144=1202.162,351.451,-75.000,-176.113,7.885,148.395
C05145=1202.158,351.699,-75.032,-176.111,7.888,148.395
C05146=1202.154,351.946,-75.065,-176.109,7.892,148.396
C05147=1202.150,352.194,-75.098,-176.108,7.894,148.396
C05148=1202.146,352.442,-75.131,-176.105,7.898,148.396
C05149=1202.141,352.690,-75.163,-176.104,7.900,148.396
C05150=1202.137,352.938,-75.197,-176.102,7.904,148.397
C05151=1202.134,353.185,-75.229,-176.100,7.907,148.397
C05152=1202.129,353.433,-75.262,-176.098,7.910,148.397
C05153=1202.125,353.681,-75.295,-176.096,7.913,148.397
C05154=1202.121,353.929,-75.328,-176.094,7.917,148.398
C05155=1202.117,354.177,-75.361,-176.092,7.919,148.398
C05156=1202.113,354.425,-75.394,-176.090,7.923,148.398
C05157=1202.108,354.672,-75.427,-176.088,7.926,148.398
C05158=1202.104,354.920,-75.461,-176.087,7.929,148.399
C05159=1202.101,355.168,-75.492,-176.085,7.932,148.399
C05160=1202.096,355.416,-75.526,-176.083,7.935,148.399
C05161=1202.092,355.663,-75.559,-176.081,7.938,148.399
C05162=1202.088,355.911,-75.592,-176.079,7.942,148.400
C05163=1202.084,356.159,-75.625,-176.077,7.944,148.400
C05164=1202.080,356.407,-75.658,-176.075,7.948,148.400
C05165=1202.076,356.654,-75.691,-176.073,7.951,148.401
C05166=1202.072,356.902,-75.724,-176.072,7.954,148.401
C05167=1202.067,357.150,-75.758,-176.070,7.957,148.401
C05168=1202.063,357.398,-75.791,-176.068,7.960,148.401
C05169=1202.059,357.645,-75.824,-176.066,7.963,148.402
C05170=1202.055,357.893,-75.857,-176.064,7.967,148.402
C05171=1202.051,358.141,-75.890,-176.063,7.969,148.402
C05172=1202.047,358.388,-75.923,-176.061,7.973,148.403
C05173=1202.043,358.636,-75.957,-176.059,7.976,148.403
C05174=1202.038,358.884,-75.990,-176.057,7.979,148.403
C05175=1202.035,359.132,-76.023,-176.055,7.982,148.403
C05176=1202.031,359.380,-76.056,-176.054,7.985,148.404
C05177=1202.027,359.628,-76.090,-176.052,7.988,148.404
C05178=1202.023,359.876,-76.123,-176.050,7.992,148.405
C05179=1202.018,360.123,-76.156,-176.048,7.995,148.405
C05180=1202.014,360.371,-76.189,-176.046,7.998,148.405
C05181=1202.010,360.619,-76.222,-176.045,8.001,148.405
C05182=1202.006,360.866,-76.256,-176.043,8.004,148.406
C05183=1202.002,361.114,-76.289,-176.041,8.007,148.406
C05184=1201.998,361.361,-76.322,-176.040,8.011,148.406
C05185=1201.993,361.609,-76.356,-176.038,8.014,148.407
C05186=1201.990,361.858,-76.390,-176.036,8.017,148.407
C05187=1201.985,362.106,-76.423,-176.034,8.020,148.407
C05188=1201.982,362.353,-76.457,-176.033,8.023,148.408
C05189=1201.978,362.600,-76.490,-176.031,8.026,148.408
C05190=1201.973,362.848,-76.523,-176.030,8.029,148.408
C05191=1201.969,363.096,-76.556,-176.027,8.033,148.409
C05192=1201.965,363.343,-76.590,-176.026,8.035,148.409
C05193=1201.961,363.591,-76.623,-176.025,8.039,148.410
C05194=1201.957,363.839,-76.657,-176.023,8.042,148.410
C05195=1201.953,364.087,-76.690,-176.021,8.045,148.410
C05196=1201.949,364.334,-76.724,-176.020,8.048,148.411
C05197=1201.945,364.582,-76.757,-176.018,8.051,148.411
C05198=1201.941,364.830,-76.791,-176.016,8.054,148.411
C05199=1201.937,365.077,-76.824,-176.015,8.058,148.412
C05200=1201.933,365.326,-76.859,-176.013,8.061,148.412
C05201=1201.928,365.573,-76.892,-176.011,8.064,148.412
C05202=1201.925,365.820,-76.926,-176.010,8.067,148.413
C05203=1201.921,366.068,-76.959,-176.008,8.070,148.413
C05204=1201.916,366.349,-76.997,-176.006,8.074,148.413
C05205=1201.911,366.630,-77.035,-176.005,8.078,148.414
C05206=1201.907,366.910,-77.073,-176.003,8.080,148.414
C05207=1201.902,367.191,-77.111,-176.002,8.084,148.415
C05208=1201.898,367.439,-77.145,-176.000,8.088,148.415
C05209=1201.894,367.686,-77.178,-175.999,8.091,148.416
C05210=1201.890,367.934,-77.213,-175.997,8.094,148.416
C05211=1201.886,368.182,-77.246,-175.995,8.097,148.416
C05212=1201.882,368.429,-77.280,-175.994,8.100,148.417
C05213=1201.877,368.677,-77.314,-175.992,8.103,148.417
C05214=1201.873,368.924,-77.347,-175.991,8.106,148.417
C05215=1201.870,369.172,-77.381,-175.989,8.110,148.418
C05216=1201.866,369.420,-77.415,-175.988,8.112,148.418
C05217=1201.861,369.667,-77.449,-175.987,8.115,148.419
C05218=1201.857,369.915,-77.482,-175.985,8.119,148.419
C05219=1201.854,370.163,-77.516,-175.984,8.122,148.419
C05220=1201.849,370.411,-77.550,-175.983,8.124,148.420
C05221=1201.845,370.658,-77.584,-175.981,8.128,148.420
C05222=1201.841,370.906,-77.617,-175.980,8.131,148.421
C05223=1201.837,371.154,-77.652,-175.978,8.134,148.421
C05224=1201.833,371.402,-77.685,-175.977,8.137,148.421
C05225=1201.829,371.649,-77.719,-175.975,8.140,148.422
C05226=1201.824,371.896,-77.754,-175.974,8.143,148.422
C05227=1201.821,372.145,-77.787,-175.973,8.147,148.423
C05228=1201.816,372.392,-77.822,-175.971,8.149,148.423
C05229=1201.812,372.640,-77.855,-175.970,8.152,148.423
C05230=1201.808,372.887,-77.889,-175.969,8.156,148.424
C05231=1201.804,373.135,-77.923,-175.968,8.159,148.425
C05232=1201.800,373.383,-77.957,-175.966,8.162,148.425
C05233=1201.796,373.630,-77.991,-175.965,8.165,148.425
C05234=1201.792,373.878,-78.025,-175.963,8.168,148.426
C05235=1201.788,374.126,-78.058,-175.962,8.171,148.426
C05236=1201.784,374.373,-78.093,-175.961,8.174,148.427
C05237=1201.780,374.620,-78.127,-175.960,8.177,148.427
C05238=1201.776,374.869,-78.161,-175.958,8.181,148.428
C05239=1201.772,375.116,-78.195,-175.957,8.183,148.428
C05240=1201.767,375.363,-78.229,-175.956,8.186,148.428
C05241=1201.764,375.611,-78.263,-175.955,8.189,148.429
C05242=1201.760,375.859,-78.297,-175.954,8.192,148.429
C05243=1201.755,376.106,-78.331,-175.952,8.196,148.430
C05244=1201.752,376.354,-78.365,-175.951,8.199,148.430
C05245=1201.747,376.602,-78.400,-175.950,8.202,148.431
C05246=1201.743,376.849,-78.433,-175.949,8.204,148.431
C05247=1201.739,377.098,-78.468,-175.948,8.207,148.432
C05248=1201.736,377.345,-78.502,-175.947,8.210,148.432
C05249=1201.731,377.592,-78.536,-175.946,8.213,148.432
C05250=1201.728,377.840,-78.570,-175.944,8.217,148.433
C05251=1201.723,378.088,-78.604,-175.943,8.220,148.434
C05252=1201.719,378.335,-78.638,-175.942,8.223,148.434
C05253=1201.715,378.583,-78.673,-175.941,8.226,148.435
C05254=1201.711,378.830,-78.707,-175.940,8.229,148.435
C05255=1201.707,379.078,-78.741,-175.939,8.231,148.435
C05256=1201.703,379.326,-78.776,-175.938,8.235,148.436
C05257=1201.699,379.573,-78.810,-175.937,8.237,148.436
C05258=1201.695,379.821,-78.845,-175.936,8.240,148.437
C05259=1201.691,380.069,-78.878,-175.935,8.243,148.437
C05260=1201.686,380.316,-78.912,-175.934,8.246,148.438
C05261=1201.683,380.564,-78.947,-175.933,8.249,148.438
C05262=1201.678,380.811,-78.981,-175.932,8.252,148.439
C05263=1201.674,381.060,-79.016,-175.931,8.255,148.439
C05264=1201.671,381.307,-79.050,-175.930,8.258,148.440
C05265=1201.666,381.554,-79.084,-175.929,8.261,148.440
C05266=1201.663,381.802,-79.118,-175.928,8.264,148.441
C05267=1201.658,382.049,-79.153,-175.927,8.267,148.441
C05268=1201.654,382.297,-79.188,-175.926,8.270,148.442
C05269=1201.650,382.544,-79.222,-175.925,8.273,148.442
C05270=1201.646,382.792,-79.256,-175.924,8.276,148.443
C05271=1201.643,383.040,-79.290,-175.923,8.279,148.443
C05272=1201.638,383.287,-79.325,-175.922,8.282,148.444
C05273=1201.634,383.535,-79.360,-175.921,8.285,148.444
C05274=1201.630,383.782,-79.393,-175.920,8.288,148.445
C05275=1201.626,384.030,-79.428,-175.919,8.291,148.445
C05276=1201.622,384.278,-79.463,-175.919,8.293,148.446
C05277=1201.618,384.525,-79.497,-175.918,8.296,148.446
C05278=1201.614,384.773,-79.531,-175.917,8.299,148.447
C05279=1201.609,385.021,-79.566,-175.916,8.302,148.447
C05280=1201.606,385.268,-79.600,-175.915,8.305,148.448
C05281=1201.602,385.516,-79.635,-175.914,8.308,148.448
C05282=1201.598,385.764,-79.669,-175.914,8.310,148.449
C05283=1201.594,386.010,-79.704,-175.913,8.313,148.449
C05284=1201.589,386.258,-79.738,-175.912,8.316,148.450
C05285=1201.585,386.506,-79.773,-175.911,8.319,148.450
C05286=1201.582,386.753,-79.807,-175.910,8.322,148.451
C05287=1201.578,387.001,-79.842,-175.909,8.324,148.451
C05288=1201.573,387.249,-79.876,-175.909,8.327,148.452
C05289=1201.570,387.496,-79.911,-175.908,8.330,148.452
C05290=1201.565,387.744,-79.945,-175.907,8.333,148.453
C05291=1201.562,387.991,-79.981,-175.906,8.335,148.453
C05292=1201.557,388.239,-80.015,-175.906,8.338,148.454
C05293=1201.554,388.487,-80.049,-175.905,8.342,148.454
C05294=1201.549,388.734,-80.084,-175.904,8.344,148.455
C05295=1201.545,388.982,-80.119,-175.904,8.347,148.455
C05296=1201.541,389.230,-80.153,-175.903,8.350,148.456
C05297=1201.538,389.477,-80.188,-175.903,8.352,148.457
C05298=1201.533,389.724,-80.223,-175.901,8.355,148.457
C05299=1201.529,389.972,-80.257,-175.901,8.358,148.458
C05300=1201.525,390.220,-80.292,-175.900,8.360,148.458
C05301=1201.522,390.467,-80.327,-175.900,8.363,148.459
C05302=1201.517,390.714,-80.361,-175.899,8.366,148.459
C05303=1201.513,390.962,-80.396,-175.898,8.368,148.460
C05304=1201.509,391.210,-80.431,-175.897,8.371,148.460
C05305=1201.506,391.457,-80.466,-175.897,8.374,148.461
C05306=1201.501,391.704,-80.500,-175.896,8.377,148.461
C05307=1201.497,391.953,-80.535,-175.896,8.379,148.462
C05308=1201.493,392.235,-80.575,-175.895,8.382,148.462
C05309=1201.488,392.518,-80.614,-175.895,8.385,148.463
C05310=1201.483,392.801,-80.654,-175.894,8.388,148.464
C05311=1201.479,393.084,-80.693,-175.893,8.392,148.464
C05312=1201.474,393.330,-80.729,-175.892,8.395,148.465
C05313=1201.471,393.578,-80.763,-175.892,8.397,148.465
C05314=1201.467,393.827,-80.798,-175.891,8.400,148.466
C05315=1201.463,394.073,-80.833,-175.891,8.402,148.466
C05316=1201.459,394.321,-80.868,-175.890,8.404,148.467
C05317=1201.454,394.569,-80.902,-175.890,8.407,148.467
C05318=1201.451,394.816,-80.938,-175.889,8.410,148.468
C05319=1201.446,395.063,-80.972,-175.889,8.413,148.468
C05320=1201.442,395.312,-81.007,-175.888,8.415,148.469
C05321=1201.439,395.558,-81.042,-175.887,8.418,148.469
C05322=1201.435,395.806,-81.076,-175.887,8.420,148.470
C05323=1201.430,396.054,-81.111,-175.886,8.423,148.471
C05324=1201.427,396.301,-81.146,-175.886,8.425,148.471
C05325=1201.423,396.549,-81.181,-175.886,8.428,148.472
C05326=1201.418,396.796,-81.216,-175.885,8.431,148.472
C05327=1201.414,397.044,-81.251,-175.885,8.433,148.473
C05328=1201.410,397.292,-81.286,-175.884,8.435,148.473
C05329=1201.407,397.539,-81.321,-175.883,8.438,148.474
C05330=1201.402,397.786,-81.355,-175.883,8.440,148.474
C05331=1201.399,398.034,-81.391,-175.883,8.443,148.475
C05332=1201.395,398.282,-81.425,-175.882,8.446,148.475
C05333=1201.390,398.529,-81.461,-175.882,8.448,148.476
C05334=1201.386,398.777,-81.495,-175.882,8.450,148.476
C05335=1201.382,399.024,-81.530,-175.881,8.453,148.477
C05336=1201.378,399.272,-81.566,-175.881,8.456,148.477
C05337=1201.374,399.519,-81.600,-175.880,8.458,148.478
C05338=1201.370,399.767,-81.636,-175.879,8.461,148.478
C05339=1201.367,400.014,-81.670,-175.879,8.463,148.479
C05340=1201.362,400.261,-81.705,-175.879,8.465,148.479
C05341=1201.358,400.509,-81.740,-175.878,8.468,148.480
C05342=1201.354,400.756,-81.775,-175.878,8.471,148.481
C05343=1201.350,401.004,-81.810,-175.877,8.473,148.481
C05344=1201.347,401.252,-81.845,-175.877,8.475,148.482
C05345=1201.342,401.499,-81.880,-175.877,8.477,148.482
C05346=1201.338,401.747,-81.915,-175.877,8.480,148.483
C05347=1201.334,401.994,-81.950,-175.875,8.483,148.483
C05348=1201.330,402.242,-81.985,-175.875,8.485,148.484
C05349=1201.326,402.490,-82.020,-175.875,8.487,148.484
C05350=1201.322,402.737,-82.055,-175.875,8.489,148.485
C05351=1201.318,402.985,-82.090,-175.875,8.492,148.485
C05352=1201.314,403.231,-82.125,-175.874,8.495,148.486
C05353=1201.310,403.479,-82.161,-175.874,8.497,148.486
C05354=1201.306,403.727,-82.196,-175.873,8.499,148.487
C05355=1201.302,403.974,-82.231,-175.873,8.502,148.487
C05356=1201.298,404.222,-82.266,-175.873,8.504,148.488
C05357=1201.294,404.469,-82.301,-175.872,8.506,148.488
C05358=1201.290,404.717,-82.336,-175.872,8.508,148.489
C05359=1201.286,404.964,-82.371,-175.872,8.510,148.489
C05360=1201.282,405.211,-82.407,-175.871,8.513,148.490
C05361=1201.278,405.459,-82.441,-175.871,8.516,148.490
C05362=1201.274,405.707,-82.477,-175.871,8.518,148.491
C05363=1201.269,405.954,-82.511,-175.870,8.520,148.492
C05364=1201.266,406.202,-82.547,-175.870,8.522,148.492
C05365=1201.262,406.449,-82.582,-175.869,8.524,148.492
C05366=1201.258,406.697,-82.617,-175.869,8.527,148.493
C05367=1201.254,406.944,-82.652,-175.869,8.529,148.493
C05368=1201.250,407.191,-82.688,-175.869,8.531,148.494
C05369=1201.246,407.439,-82.722,-175.868,8.534,148.495
C05370=1201.242,407.687,-82.758,-175.868,8.536,148.495
C05371=1201.238,407.933,-82.793,-175.868,8.538,148.496
C05372=1201.234,408.181,-82.828,-175.868,8.540,148.496
C05373=1201.230,408.429,-82.864,-175.867,8.542,148.496
C05374=1201.226,408.676,-82.899,-175.867,8.545,148.497
C05375=1201.222,408.924,-82.934,-175.867,8.547,148.497
C05376=1201.218,409.171,-82.969,-175.866,8.549,148.498
C05377=1201.214,409.418,-83.004,-175.866,8.551,148.499
C05378=1201.210,409.666,-83.039,-175.866,8.554,148.499
C05379=1201.206,409.914,-83.075,-175.866,8.556,148.500
C05380=1201.202,410.161,-83.110,-175.865,8.558,148.500
C05381=1201.198,410.409,-83.145,-175.865,8.560,148.500
C05382=1201.194,410.656,-83.180,-175.865,8.562,148.501
C05383=1201.190,410.903,-83.215,-175.864,8.565,148.502
C05384=1201.186,411.151,-83.250,-175.864,8.567,148.502
C05385=1201.183,411.399,-83.286,-175.864,8.569,148.503
C05386=1201.178,411.645,-83.321,-175.863,8.571,148.503
C05387=1201.175,411.893,-83.357,-175.863,8.573,148.503
C05388=1201.170,412.141,-83.392,-175.863,8.576,148.504
C05389=1201.166,412.389,-83.428,-175.863,8.578,148.505
C05390=1201.162,412.636,-83.463,-175.862,8.580,148.505
C05391=1201.158,412.883,-83.498,-175.862,8.583,148.506
C05392=1201.154,413.131,-83.533,-175.861,8.584,148.506
C05393=1201.150,413.378,-83.568,-175.861,8.587,148.506
C05394=1201.146,413.626,-83.604,-175.862,8.588,148.507
C05395=1201.143,413.873,-83.639,-175.861,8.590,148.507
C05396=1201.138,414.121,-83.674,-175.861,8.593,148.508
C05397=1201.135,414.368,-83.709,-175.860,8.595,148.508
C05398=1201.131,414.616,-83.745,-175.860,8.597,148.509
C05399=1201.126,414.863,-83.781,-175.860,8.599,148.509
C05400=1201.122,415.110,-83.816,-175.860,8.601,148.510
C05401=1201.118,415.358,-83.851,-175.859,8.604,148.510
C05402=1201.115,415.606,-83.887,-175.859,8.606,148.511
C05403=1201.110,415.853,-83.922,-175.859,8.607,148.511
C05404=1201.105,416.165,-83.966,-175.858,8.610,148.512
C05405=1201.101,416.477,-84.011,-175.859,8.613,148.513
C05406=1201.100,416.789,-84.056,-175.858,8.615,148.513
C05407=1201.103,417.101,-84.099,-175.858,8.617,148.514
C05408=1200.681,417.101,-84.138,-175.861,8.629,148.517
C05409=1200.679,416.786,-84.093,-175.862,8.626,148.517
C05410=1200.680,416.472,-84.049,-175.861,8.623,148.516
C05411=1200.684,416.157,-84.003,-175.862,8.621,148.515
C05412=1200.689,415.842,-83.958,-175.862,8.618,148.515
C05413=1200.693,415.594,-83.924,-175.862,8.616,148.514
C05414=1200.697,415.347,-83.888,-175.862,8.614,148.514
C05415=1200.700,415.099,-83.853,-175.863,8.612,148.514
C05416=1200.705,414.853,-83.817,-175.863,8.610,148.513
C05417=1200.708,414.605,-83.782,-175.863,8.608,148.513
C05418=1200.713,414.357,-83.746,-175.864,8.605,148.512
C05419=1200.717,414.109,-83.711,-175.864,8.603,148.511
C05420=1200.721,413.862,-83.676,-175.865,8.601,148.511
C05421=1200.725,413.615,-83.640,-175.864,8.600,148.511
C05422=1200.728,413.367,-83.605,-175.864,8.597,148.510
C05423=1200.733,413.120,-83.570,-175.865,8.595,148.510
C05424=1200.737,412.872,-83.535,-175.865,8.593,148.509
C05425=1200.740,412.625,-83.499,-175.866,8.591,148.509
C05426=1200.744,412.378,-83.464,-175.866,8.589,148.508
C05427=1200.748,412.130,-83.429,-175.866,8.586,148.508
C05428=1200.753,411.882,-83.393,-175.866,8.584,148.507
C05429=1200.757,411.635,-83.358,-175.866,8.582,148.507
C05430=1200.761,411.388,-83.322,-175.867,8.580,148.506
C05431=1200.765,411.140,-83.287,-175.867,8.578,148.506
C05432=1200.769,410.893,-83.252,-175.868,8.575,148.505
C05433=1200.773,410.646,-83.217,-175.868,8.573,148.505
C05434=1200.777,410.397,-83.182,-175.868,8.571,148.504
C05435=1200.780,410.150,-83.146,-175.868,8.569,148.504
C05436=1200.785,409.903,-83.111,-175.869,8.566,148.503
C05437=1200.788,409.656,-83.076,-175.868,8.565,148.503
C05438=1200.792,409.407,-83.041,-175.869,8.563,148.502
C05439=1200.796,409.161,-83.006,-175.869,8.561,148.502
C05440=1200.800,408.913,-82.970,-175.869,8.558,148.501
C05441=1200.804,408.665,-82.935,-175.870,8.556,148.501
C05442=1200.808,408.418,-82.900,-175.870,8.554,148.500
C05443=1200.812,408.171,-82.864,-175.870,8.552,148.500
C05444=1200.816,407.923,-82.830,-175.871,8.548,148.499
C05445=1200.820,407.676,-82.794,-175.871,8.546,148.499
C05446=1200.825,407.428,-82.758,-175.872,8.544,148.498
C05447=1200.829,407.181,-82.724,-175.872,8.542,148.498
C05448=1200.833,406.933,-82.688,-175.872,8.540,148.497
C05449=1200.837,406.686,-82.653,-175.872,8.537,148.497
C05450=1200.841,406.438,-82.618,-175.873,8.535,148.496
C05451=1200.845,406.191,-82.583,-175.873,8.533,148.496
C05452=1200.848,405.943,-82.547,-175.873,8.531,148.495
C05453=1200.853,405.696,-82.513,-175.873,8.528,148.494
C05454=1200.857,405.448,-82.477,-175.874,8.526,148.494
C05455=1200.861,405.200,-82.442,-175.874,8.524,148.494
C05456=1200.865,404.953,-82.407,-175.874,8.522,148.493
C05457=1200.869,404.706,-82.372,-175.875,8.520,148.493
C05458=1200.873,404.458,-82.337,-175.875,8.516,148.492
C05459=1200.877,404.211,-82.302,-175.876,8.514,148.491
C05460=1200.881,403.963,-82.267,-175.876,8.512,148.491
C05461=1200.885,403.716,-82.232,-175.876,8.510,148.490
C05462=1200.889,403.468,-82.197,-175.876,8.507,148.490
C05463=1200.893,403.220,-82.161,-175.877,8.505,148.489
C05464=1200.896,402.974,-82.127,-175.877,8.503,148.489
C05465=1200.900,402.726,-82.092,-175.878,8.500,148.488
C05466=1200.904,402.479,-82.057,-175.878,8.498,148.488
C05467=1200.908,402.231,-82.022,-175.879,8.495,148.487
C05468=1200.912,401.983,-81.986,-175.879,8.493,148.487
C05469=1200.917,401.736,-81.952,-175.879,8.491,148.486
C05470=1200.920,401.488,-81.916,-175.879,8.489,148.486
C05471=1200.924,401.240,-81.881,-175.880,8.486,148.485
